KUKA KRL program: MyProgram_236().src

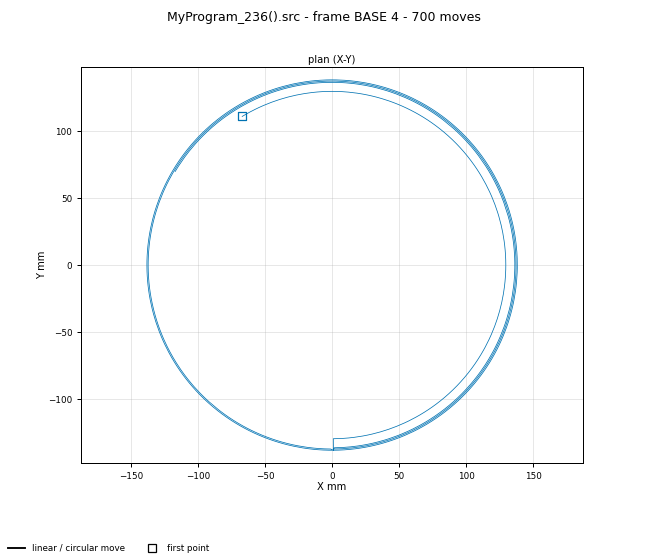
[picture p0: tool path of MyProgram_236().src in frame BASE 4, 700 of 700 moves have a stored position in this frame; points joined in program order, loops and branches not executed]
&ACCESS RVP
&REL 1
&PARAM TEMPLATE = C:\KRC\Roboter\Template\vorgabe
&PARAM EDITMASK = *
DEF MyProgram_236()
; ---- Setting reference (Base) ----
$BASE = BASE_DATA[4]

; --------------------------
; ---- Setting tool (TCP) ----
$TOOL = TOOL_DATA[3]
; --------------------------

$VEL.CP = VEL_APROX_PRINT
Startdeposition()
$VEL.CP = VEL_PRINT
LIN {X -67.1203,Y 110.906,Z 159,A 119.8664,B 14.7738,C -0.2462,E1 14.6942,E2 329.6728} C_DIS
LIN {X -63.8698,Y 112.81,Z 159,A 118.1875,B 14.7738,C -0.2484,E1 14.6982,E2 331.3516} C_DIS
LIN {X -61.0916,Y 114.338,Z 159,A 116.7775,B 14.7738,C -0.2503,E1 14.7017,E2 332.7612} C_DIS
LIN {X -57.3512,Y 116.2566,Z 159,A 114.9162,B 14.7737,C -0.2529,E1 14.7063,E2 334.6209} C_DIS
LIN {X -54.4896,Y 117.6251,Z 159,A 113.4128,B 14.7737,C -0.2521,E1 14.7102,E2 336.1345} C_DIS
LIN {X -51.0857,Y 119.1435,Z 159,A 111.8471,B 14.7737,C -0.2564,E1 14.7141,E2 337.6895} C_DIS
LIN {X -48.1337,Y 120.3663,Z 159,A 110.4314,B 14.7736,C -0.2581,E1 14.7178,E2 339.1043} C_DIS
LIN {X -45.1664,Y 121.5109,Z 159,A 109.0181,B 14.7736,C -0.2595,E1 14.7215,E2 340.5173} C_DIS
LIN {X -42.1522,Y 122.5891,Z 159,A 107.6016,B 14.7736,C -0.261,E1 14.7252,E2 341.9327} C_DIS
LIN {X -39.1386,Y 123.5843,Z 159,A 106.1946,B 14.7736,C -0.2623,E1 14.7289,E2 343.3391} C_DIS
LIN {X -36.1004,Y 124.5058,Z 159,A 104.7875,B 14.7736,C -0.2635,E1 14.7327,E2 344.7455} C_DIS
LIN {X -33.0403,Y 125.3527,Z 159,A 103.3786,B 14.7735,C -0.2646,E1 14.7365,E2 346.1539} C_DIS
LIN {X -29.9406,Y 126.1293,Z 159,A 101.9667,B 14.7735,C -0.2657,E1 14.7403,E2 347.5647} C_DIS
LIN {X -26.8488,Y 126.8237,Z 159,A 100.5599,B 14.7735,C -0.2665,E1 14.7442,E2 348.9712} C_DIS
LIN {X -24.2125,Y 127.3523,Z 159,A 99.3725,B 14.7735,C -0.2674,E1 14.7474,E2 350.1576} C_DIS
LIN {X -20.8059,Y 127.9541,Z 159,A 97.868,B 14.7735,C -0.269,E1 14.7516,E2 351.6584} C_DIS
LIN {X -18.0217,Y 128.3752,Z 159,A 96.6198,B 14.7734,C -0.2695,E1 14.755,E2 352.9061} C_DIS
LIN {X -14.8341,Y 128.7831,Z 159,A 95.0397,B 14.7734,C -0.2656,E1 14.7594,E2 354.5036} C_DIS
LIN {X -11.1216,Y 129.1559,Z 159,A 93.509,B 14.7734,C -0.2696,E1 14.7636,E2 356.0199} C_DIS
LIN {X -7.5683,Y 129.4132,Z 159,A 91.939,B 14.7734,C -0.2702,E1 14.768,E2 357.5884} C_DIS
LIN {X -3.731,Y 129.5801,Z 159,A 90.2362,B 14.7734,C -0.2704,E1 14.7728,E2 359.2909} C_DIS
LIN {X 0.0023,Y 129.6358,Z 159,A 88.562,B 14.7734,C -0.2699,E1 14.7774,E2 360.9671} C_DIS
LIN {X 3.733,Y 129.5801,Z 159,A 86.8871,B 14.7734,C -0.2692,E1 14.7821,E2 362.6441} C_DIS
LIN {X 7.9541,Y 129.3894,Z 159,A 84.9994,B 14.7734,C -0.2685,E1 14.7874,E2 364.5334} C_DIS
LIN {X 12.1572,Y 129.0626,Z 159,A 83.138,B 14.7734,C -0.2682,E1 14.7926,E2 366.3939} C_DIS
LIN {X 16.0012,Y 128.6439,Z 159,A 81.5164,B 14.7734,C -0.2703,E1 14.797,E2 368.005} C_DIS
LIN {X 18.6052,Y 128.2918,Z 159,A 80.3418,B 14.7734,C -0.2696,E1 14.8003,E2 369.1807} C_DIS
LIN {X 22.1957,Y 127.7209,Z 159,A 78.5869,B 14.7734,C -0.2645,E1 14.8052,E2 370.9521} C_DIS
LIN {X 26.3286,Y 126.9326,Z 159,A 76.8852,B 14.7734,C -0.2683,E1 14.8098,E2 372.6354} C_DIS
LIN {X 29.4247,Y 126.2511,Z 159,A 75.486,B 14.7734,C -0.2676,E1 14.8136,E2 374.0341} C_DIS
LIN {X 33.0382,Y 125.3533,Z 159,A 73.7666,B 14.7734,C -0.2643,E1 14.8183,E2 375.7616} C_DIS
LIN {X 37.1039,Y 124.212,Z 159,A 71.979,B 14.7734,C -0.2653,E1 14.823,E2 377.5401} C_DIS
LIN {X 40.1416,Y 123.2639,Z 159,A 70.5796,B 14.7734,C -0.2643,E1 14.8268,E2 378.9385} C_DIS
LIN {X 42.6971,Y 122.4002,Z 159,A 69.3347,B 14.7735,C -0.2617,E1 14.8301,E2 380.1893} C_DIS
LIN {X 45.6848,Y 121.3167,Z 159,A 67.9319,B 14.7735,C -0.2604,E1 14.8337,E2 381.5919} C_DIS
LIN {X 49.089,Y 119.9813,Z 159,A 66.3714,B 14.7735,C -0.2604,E1 14.8378,E2 383.146} C_DIS
LIN {X 52.0319,Y 118.7345,Z 159,A 64.8389,B 14.7736,C -0.2552,E1 14.8417,E2 384.6923} C_DIS
LIN {X 55.4342,Y 117.1839,Z 159,A 63.328,B 14.7736,C -0.2576,E1 14.8455,E2 386.1871} C_DIS
LIN {X 58.7836,Y 115.539,Z 159,A 61.6551,B 14.7736,C -0.2548,E1 14.8497,E2 387.8628} C_DIS
LIN {X 62.0192,Y 113.8372,Z 159,A 60.0736,B 14.7736,C -0.2537,E1 14.8536,E2 389.4408} C_DIS
LIN {X 64.7903,Y 112.2832,Z 159,A 58.5716,B 14.7738,C -0.2487,E1 14.8573,E2 390.9543} C_DIS
LIN {X 68.0623,Y 110.3309,Z 159,A 56.8912,B 14.7738,C -0.2463,E1 14.8613,E2 392.6346} C_DIS
LIN {X 71.5703,Y 108.0883,Z 159,A 55.1642,B 14.7738,C -0.2469,E1 14.8653,E2 394.3491} C_DIS
LIN {X 74.1944,Y 106.3038,Z 159,A 53.7715,B 14.7738,C -0.2449,E1 14.8685,E2 395.7411} C_DIS
LIN {X 77.2242,Y 104.1238,Z 159,A 51.9984,B 14.7739,C -0.2383,E1 14.8725,E2 397.529} C_DIS
LIN {X 80.4688,Y 101.6374,Z 159,A 50.1936,B 14.7739,C -0.2352,E1 14.8765,E2 399.3342} C_DIS
LIN {X 83.8675,Y 98.8511,Z 159,A 48.359,B 14.7739,C -0.2349,E1 14.8804,E2 401.1572} C_DIS
LIN {X 86.6751,Y 96.399,Z 159,A 46.6678,B 14.774,C -0.2304,E1 14.884,E2 402.8541} C_DIS
LIN {X 89.7611,Y 93.5323,Z 159,A 44.8758,B 14.774,C -0.2289,E1 14.8876,E2 404.639} C_DIS
LIN {X 92.742,Y 90.5774,Z 159,A 42.9905,B 14.7741,C -0.2241,E1 14.8913,E2 406.5288} C_DIS
LIN {X 95.5533,Y 87.6064,Z 159,A 41.2364,B 14.7741,C -0.2219,E1 14.8946,E2 408.2777} C_DIS
LIN {X 98.3326,Y 84.4748,Z 159,A 39.347,B 14.7742,C -0.2166,E1 14.8981,E2 410.1727} C_DIS
LIN {X 101.04,Y 81.2173,Z 159,A 37.4829,B 14.7743,C -0.2127,E1 14.9014,E2 412.0371} C_DIS
LIN {X 103.7073,Y 77.7832,Z 159,A 35.5408,B 14.7743,C -0.2075,E1 14.9047,E2 413.9828} C_DIS
LIN {X 105.9847,Y 74.6493,Z 159,A 33.989,B 14.7743,C -0.2086,E1 14.9072,E2 415.5174} C_DIS
LIN {X 107.7826,Y 72.0291,Z 159,A 32.599,B 14.7744,C -0.2056,E1 14.9094,E2 416.9066} C_DIS
LIN {X 109.8271,Y 68.8726,Z 159,A 30.8417,B 14.7744,C -0.1984,E1 14.912,E2 418.6763} C_DIS
LIN {X 111.7248,Y 65.7484,Z 159,A 29.2525,B 14.7745,C -0.1952,E1 14.9143,E2 420.2637} C_DIS
LIN {X 113.5698,Y 62.5083,Z 159,A 27.7539,B 14.7745,C -0.1958,E1 14.9163,E2 421.7464} C_DIS
LIN {X 114.8093,Y 60.1962,Z 159,A 26.5652,B 14.7745,C -0.1918,E1 14.9179,E2 422.9394} C_DIS
LIN {X 116.2491,Y 57.3666,Z 159,A 25.1756,B 14.7746,C -0.1885,E1 14.9196,E2 424.3286} C_DIS
LIN {X 117.6203,Y 54.5,Z 159,A 23.6885,B 14.7747,C -0.1821,E1 14.9214,E2 425.8266} C_DIS
LIN {X 119.1501,Y 51.0705,Z 159,A 22.1376,B 14.7747,C -0.1811,E1 14.9231,E2 427.3664} C_DIS
LIN {X 120.3664,Y 48.1335,Z 159,A 20.7467,B 14.7747,C -0.1777,E1 14.9246,E2 428.757} C_DIS
LIN {X 121.5105,Y 45.1674,Z 159,A 19.3557,B 14.7747,C -0.1743,E1 14.926,E2 430.1477} C_DIS
LIN {X 122.5834,Y 42.1688,Z 159,A 17.9628,B 14.7748,C -0.1708,E1 14.9273,E2 431.5403} C_DIS
LIN {X 123.5841,Y 39.1391,Z 159,A 16.5673,B 14.7748,C -0.1673,E1 14.9285,E2 432.9355} C_DIS
LIN {X 124.4063,Y 36.44,Z 159,A 15.2755,B 14.7749,C -0.1623,E1 14.9295,E2 434.2338} C_DIS
LIN {X 125.3524,Y 33.0414,Z 159,A 13.7909,B 14.7749,C -0.1602,E1 14.9306,E2 435.7114} C_DIS
LIN {X 126.124,Y 29.9624,Z 159,A 12.4206,B 14.7749,C -0.1572,E1 14.9315,E2 437.0794} C_DIS
LIN {X 126.8601,Y 26.6802,Z 159,A 10.9379,B 14.775,C -0.153,E1 14.9324,E2 438.5633} C_DIS
LIN {X 127.3533,Y 24.2074,Z 159,A 9.8335,B 14.775,C -0.1501,E1 14.933,E2 439.6677} C_DIS
LIN {X 127.9849,Y 20.6214,Z 159,A 8.2534,B 14.775,C -0.1462,E1 14.9337,E2 441.2463} C_DIS
LIN {X 128.3792,Y 17.9938,Z 159,A 7.0773,B 14.7751,C -0.1427,E1 14.9342,E2 442.4238} C_DIS
LIN {X 128.7823,Y 14.841,Z 159,A 5.5559,B 14.7751,C -0.1347,E1 14.9347,E2 443.9605} C_DIS
LIN {X 129.1554,Y 11.1276,Z 159,A 3.9869,B 14.7752,C -0.1324,E1 14.9351,E2 445.522} C_DIS
LIN {X 129.4343,Y 7.2235,Z 159,A 2.3652,B 14.7752,C -0.1308,E1 14.9354,E2 447.1332} C_DIS
LIN {X 129.5799,Y 3.7378,Z 159,A 0.8063,B 14.7752,C -0.1256,E1 14.9356,E2 448.6959} C_DIS
LIN {X 129.636,Y 0.0053,Z 159,A -0.8546,B 14.7753,C -0.1202,E1 14.9356,E2 450.3602} C_DIS
LIN {X 129.5905,Y -3.3568,Z 159,A -2.4308,B 14.7753,C -0.1128,E1 14.9356,E2 451.9486} C_DIS
LIN {X 129.3897,Y -7.9495,Z 159,A -4.3756,B 14.7754,C -0.1096,E1 14.9352,E2 453.8858} C_DIS
LIN {X 129.0632,Y -12.1507,Z 159,A -6.1534,B 14.7754,C -0.1067,E1 14.9348,E2 455.656} C_DIS
LIN {X 128.6351,Y -16.0754,Z 159,A -7.8536,B 14.7754,C -0.1029,E1 14.9343,E2 457.3533} C_DIS
LIN {X 128.2236,Y -19.0827,Z 159,A -9.2075,B 14.7754,C -0.0985,E1 14.9337,E2 458.7104} C_DIS
LIN {X 127.8138,Y -21.6469,Z 159,A -10.418,B 14.7755,C -0.093,E1 14.9332,E2 459.9295} C_DIS
LIN {X 127.1942,Y -25.0399,Z 159,A -11.8339,B 14.7755,C -0.092,E1 14.9324,E2 461.3348} C_DIS
LIN {X 126.6015,Y -27.8778,Z 159,A -13.11,B 14.7755,C -0.0884,E1 14.9317,E2 462.6119} C_DIS
LIN {X 125.9172,Y -30.8204,Z 159,A -14.4371,B 14.7755,C -0.0847,E1 14.9308,E2 463.9398} C_DIS
LIN {X 125.0892,Y -34.0284,Z 159,A -15.8607,B 14.7755,C -0.0817,E1 14.9298,E2 465.3605} C_DIS
LIN {X 124.2104,Y -37.1093,Z 159,A -17.2862,B 14.7756,C -0.0772,E1 14.9287,E2 466.789} C_DIS
LIN {X 123.2639,Y -40.1415,Z 159,A -18.6777,B 14.7756,C -0.0736,E1 14.9275,E2 468.1808} C_DIS
LIN {X 122.4011,Y -42.6947,Z 159,A -19.9406,B 14.7756,C -0.0678,E1 14.9264,E2 469.4537} C_DIS
LIN {X 121.282,Y -45.7774,Z 159,A -21.336,B 14.7756,C -0.0654,E1 14.925,E2 470.8447} C_DIS
LIN {X 119.9587,Y -49.145,Z 159,A -22.8797,B 14.7756,C -0.0626,E1 14.9234,E2 472.3841} C_DIS
LIN {X 118.8209,Y -51.8319,Z 159,A -24.1799,B 14.7756,C -0.0587,E1 14.922,E2 473.6871} C_DIS
LIN {X 117.1943,Y -55.4124,Z 159,A -25.8759,B 14.7756,C -0.0552,E1 14.92,E2 475.3804} C_DIS
LIN {X 115.7914,Y -58.2877,Z 159,A -27.2678,B 14.7757,C -0.052,E1 14.9183,E2 476.7716} C_DIS
LIN {X 114.3285,Y -61.1093,Z 159,A -28.5712,B 14.7757,C -0.0515,E1 14.9166,E2 478.0649} C_DIS
LIN {X 113.0667,Y -63.413,Z 159,A -29.9152,B 14.7757,C -0.0423,E1 14.9147,E2 479.432} C_DIS
LIN {X 110.8982,Y -67.1332,Z 159,A -31.7839,B 14.7757,C -0.0384,E1 14.9121,E2 481.2991} C_DIS
LIN {X 108.6614,Y -70.6965,Z 159,A -33.5454,B 14.7757,C -0.0367,E1 14.9095,E2 483.0515} C_DIS
LIN {X 106.5523,Y -73.8374,Z 159,A -35.2973,B 14.7757,C -0.0298,E1 14.9067,E2 484.8149} C_DIS
LIN {X 104.1116,Y -77.2405,Z 159,A -37.1373,B 14.7757,C -0.0255,E1 14.9037,E2 486.656} C_DIS
LIN {X 101.5297,Y -80.6041,Z 159,A -38.9905,B 14.7757,C -0.0216,E1 14.9005,E2 488.5091} C_DIS
LIN {X 98.8199,Y -83.9042,Z 159,A -40.8594,B 14.7757,C -0.0176,E1 14.8971,E2 490.3782} C_DIS
LIN {X 96.0345,Y -87.0784,Z 159,A -42.7041,B 14.7757,C -0.014,E1 14.8937,E2 492.2226} C_DIS
LIN {X 93.3312,Y -89.9702,Z 159,A -44.4989,B 14.7757,C -0.0085,E1 14.8902,E2 494.0249} C_DIS
LIN {X 90.133,Y -93.1735,Z 159,A -46.4359,B 14.7757,C -0.0061,E1 14.8864,E2 495.9568} C_DIS
LIN {X 87.0427,Y -96.0669,Z 159,A -48.287,B 14.7758,C -0.0027,E1 14.8826,E2 497.8078} C_DIS
LIN {X 84.0655,Y -98.6827,Z 159,A -49.989,B 14.7758,C -0.0007,E1 14.879,E2 499.506} C_DIS
LIN {X 80.9868,Y -101.2251,Z 159,A -51.8385,B 14.7758,C 0.0056,E1 14.875,E2 501.3675} C_DIS
LIN {X 77.6558,Y -103.8024,Z 159,A -53.6478,B 14.7758,C 0.0076,E1 14.871,E2 503.1727} C_DIS
LIN {X 74.6416,Y -105.9902,Z 159,A -55.1713,B 14.7758,C 0.0067,E1 14.8675,E2 504.6837} C_DIS
LIN {X 72.0229,Y -107.7867,Z 159,A -56.5633,B 14.7758,C 0.0089,E1 14.8643,E2 506.0757} C_DIS
LIN {X 68.9171,Y -109.799,Z 159,A -58.3045,B 14.7758,C 0.0151,E1 14.8602,E2 507.8312} C_DIS
LIN {X 65.7525,Y -111.7224,Z 159,A -59.896,B 14.7758,C 0.0164,E1 14.8564,E2 509.4191} C_DIS
LIN {X 62.5084,Y -113.5697,Z 159,A -61.4627,B 14.7758,C 0.0164,E1 14.8526,E2 510.9776} C_DIS
LIN {X 59.5138,Y -115.1672,Z 159,A -62.9484,B 14.7758,C 0.0183,E1 14.8489,E2 512.4632} C_DIS
LIN {X 57.2074,Y -116.3276,Z 159,A -64.0735,B 14.7758,C 0.0195,E1 14.8461,E2 513.5874} C_DIS
LIN {X 54.0617,Y -117.8229,Z 159,A -65.6278,B 14.7758,C 0.0221,E1 14.8422,E2 515.145} C_DIS
LIN {X 51.0647,Y -119.1526,Z 159,A -67.0629,B 14.7758,C 0.0236,E1 14.8385,E2 516.5798} C_DIS
LIN {X 48.1302,Y -120.3678,Z 159,A -68.4596,B 14.7758,C 0.0252,E1 14.8349,E2 517.9769} C_DIS
LIN {X 45.1639,Y -121.5118,Z 159,A -69.8579,B 14.7758,C 0.0267,E1 14.8312,E2 519.3757} C_DIS
LIN {X 42.1715,Y -122.5825,Z 159,A -71.2646,B 14.7758,C 0.0283,E1 14.8275,E2 520.7837} C_DIS
LIN {X 39.097,Y -123.5976,Z 159,A -72.6797,B 14.7758,C 0.0294,E1 14.8237,E2 522.1982} C_DIS
LIN {X 36.0775,Y -124.5125,Z 159,A -74.0689,B 14.7758,C 0.0306,E1 14.82,E2 523.588} C_DIS
LIN {X 33.0288,Y -125.3558,Z 159,A -75.4487,B 14.7758,C 0.0314,E1 14.8163,E2 524.9666} C_DIS
LIN {X 29.9586,Y -126.1249,Z 159,A -76.8546,B 14.7758,C 0.0328,E1 14.8125,E2 526.3745} C_DIS
LIN {X 26.3447,Y -126.9293,Z 159,A -78.5984,B 14.7758,C 0.0374,E1 14.8077,E2 528.1321} C_DIS
LIN {X 22.7058,Y -127.6296,Z 159,A -80.1843,B 14.7758,C 0.0369,E1 14.8034,E2 529.713} C_DIS
LIN {X 19.5724,Y -128.1478,Z 159,A -81.5205,B 14.7758,C 0.0357,E1 14.7997,E2 531.0423} C_DIS
LIN {X 16.4157,Y -128.5908,Z 159,A -83.0436,B 14.7758,C 0.04,E1 14.7954,E2 532.5797} C_DIS
LIN {X 12.1492,Y -129.0633,Z 159,A -84.886,B 14.7758,C 0.0392,E1 14.7903,E2 534.4168} C_DIS
LIN {X 7.9488,Y -129.3898,Z 159,A -86.7504,B 14.7758,C 0.0399,E1 14.7851,E2 536.2825} C_DIS
LIN {X 3.7245,Y -129.5803,Z 159,A -88.5546,B 14.7758,C 0.0385,E1 14.7801,E2 538.0802} C_DIS
LIN {X 0.8939,Y -129.6275,Z 159,A -89.3751,B 14.7758,C 0.0257,E1 14.778,E2 538.8503} C_DIS
Enddeposition()
LIN {X 0.9745,Y -138.2214,Z 160,A -92.2372,B 24.9707,C -1.2506,E1 25.0023,E2 538.9144} C_DIS
Startdeposition()
$VEL.CP = VEL_PRINT
LIN {X 4.9672,Y -138.1363,Z 160,A -90.5146,B 24.9705,C -1.2549,E1 25.0072,E2 537.182} C_DIS
LIN {X 8.9652,Y -137.9346,Z 160,A -88.7661,B 24.9702,C -1.2605,E1 25.0121,E2 535.4208} C_DIS
LIN {X 12.9848,Y -137.6138,Z 160,A -87.2521,B 24.9706,C -1.2526,E1 25.0162,E2 533.9264} C_DIS
LIN {X 17.0609,Y -137.1696,Z 160,A -85.4986,B 24.9704,C -1.2567,E1 25.0211,E2 532.1646} C_DIS
LIN {X 20.739,Y -136.6607,Z 160,A -83.946,B 24.9704,C -1.2585,E1 25.0254,E2 530.609} C_DIS
LIN {X 24.3768,Y -136.0582,Z 160,A -82.4644,B 24.9704,C -1.2571,E1 25.0295,E2 529.1323} C_DIS
LIN {X 27.7328,Y -135.4141,Z 160,A -81.0374,B 24.9704,C -1.259,E1 25.0334,E2 527.7026} C_DIS
LIN {X 31.1838,Y -134.6618,Z 160,A -79.4483,B 24.9699,C -1.2674,E1 25.0378,E2 526.0957} C_DIS
LIN {X 34.8431,Y -133.7633,Z 160,A -78.028,B 24.9702,C -1.261,E1 25.0416,E2 524.6926} C_DIS
LIN {X 38.2167,Y -132.838,Z 160,A -76.5857,B 24.9702,C -1.2622,E1 25.0455,E2 523.25} C_DIS
LIN {X 41.4498,Y -131.8649,Z 160,A -75.1438,B 24.97,C -1.2663,E1 25.0493,E2 521.801} C_DIS
LIN {X 44.7534,Y -130.7801,Z 160,A -73.6382,B 24.9697,C -1.2718,E1 25.0533,E2 520.2853} C_DIS
LIN {X 48.3409,Y -129.4959,Z 160,A -72.1957,B 24.97,C -1.2662,E1 25.0571,E2 518.8591} C_DIS
LIN {X 51.4463,Y -128.294,Z 160,A -70.8247,B 24.97,C -1.2676,E1 25.0606,E2 517.4876} C_DIS
LIN {X 54.8596,Y -126.8716,Z 160,A -69.2999,B 24.9698,C -1.2695,E1 25.0646,E2 515.962} C_DIS
LIN {X 57.9395,Y -125.495,Z 160,A -67.8796,B 24.9697,C -1.273,E1 25.0682,E2 514.5371} C_DIS
LIN {X 60.4907,Y -124.2875,Z 160,A -66.6861,B 24.9695,C -1.2762,E1 25.0712,E2 513.3391} C_DIS
LIN {X 63.6062,Y -122.7223,Z 160,A -65.2643,B 24.9695,C -1.2774,E1 25.0747,E2 511.9184} C_DIS
LIN {X 66.6673,Y -121.0872,Z 160,A -63.7025,B 24.969,C -1.287,E1 25.0786,E2 510.3384} C_DIS
LIN {X 70.4482,Y -118.9273,Z 160,A -61.8999,B 24.9688,C -1.2903,E1 25.083,E2 508.5336} C_DIS
LIN {X 74.2885,Y -116.5668,Z 160,A -60.0462,B 24.9687,C -1.2931,E1 25.0873,E2 506.6792} C_DIS
LIN {X 77.8899,Y -114.1921,Z 160,A -58.3083,B 24.9687,C -1.2938,E1 25.0914,E2 504.9453} C_DIS
LIN {X 81.4971,Y -111.6464,Z 160,A -56.5752,B 24.9687,C -1.2921,E1 25.0953,E2 503.2223} C_DIS
LIN {X 84.31,Y -109.5377,Z 160,A -54.9752,B 24.9682,C -1.3036,E1 25.0989,E2 501.6011} C_DIS
LIN {X 87.8225,Y -106.7423,Z 160,A -53.1459,B 24.9681,C -1.306,E1 25.1028,E2 499.773} C_DIS
LIN {X 91.2002,Y -103.8712,Z 160,A -51.2962,B 24.9678,C -1.311,E1 25.1068,E2 497.9188} C_DIS
LIN {X 94.3975,Y -100.9737,Z 160,A -49.6476,B 24.968,C -1.3073,E1 25.1101,E2 496.2857} C_DIS
LIN {X 97.053,Y -98.4244,Z 160,A -48.142,B 24.9679,C -1.3099,E1 25.1131,E2 494.7802} C_DIS
LIN {X 99.5318,Y -95.9169,Z 160,A -46.6892,B 24.9677,C -1.3131,E1 25.116,E2 493.3261} C_DIS
LIN {X 101.9451,Y -93.3477,Z 160,A -45.2383,B 24.9675,C -1.3163,E1 25.1187,E2 491.874} C_DIS
LIN {X 104.2139,Y -90.8074,Z 160,A -43.7946,B 24.9673,C -1.3219,E1 25.1214,E2 490.4236} C_DIS
LIN {X 106.6121,Y -87.9797,Z 160,A -42.291,B 24.9672,C -1.3241,E1 25.1241,E2 488.9217} C_DIS
LIN {X 108.8159,Y -85.2388,Z 160,A -40.858,B 24.967,C -1.3267,E1 25.1266,E2 487.4893} C_DIS
LIN {X 110.943,Y -82.4511,Z 160,A -39.414,B 24.9669,C -1.3302,E1 25.129,E2 486.044} C_DIS
LIN {X 113.1108,Y -79.4515,Z 160,A -37.8654,B 24.9666,C -1.3354,E1 25.1315,E2 484.4905} C_DIS
LIN {X 115.116,Y -76.5173,Z 160,A -36.4114,B 24.9664,C -1.3385,E1 25.1338,E2 483.0364} C_DIS
LIN {X 117.4083,Y -72.9508,Z 160,A -34.6661,B 24.9662,C -1.343,E1 25.1364,E2 481.2895} C_DIS
LIN {X 119.2406,Y -69.9157,Z 160,A -33.2242,B 24.9661,C -1.3457,E1 25.1384,E2 479.8484} C_DIS
LIN {X 121.2665,Y -66.34,Z 160,A -31.487,B 24.9657,C -1.3528,E1 25.1408,E2 478.1035} C_DIS
LIN {X 123.0416,Y -62.9827,Z 160,A -29.9644,B 24.9657,C -1.3547,E1 25.1428,E2 476.5846} C_DIS
LIN {X 124.5999,Y -59.8407,Z 160,A -28.4957,B 24.9654,C -1.36,E1 25.1446,E2 475.1112} C_DIS
LIN {X 126.1424,Y -56.5163,Z 160,A -27.0475,B 24.9654,C -1.3606,E1 25.1463,E2 473.6694} C_DIS
LIN {X 127.6265,Y -53.0803,Z 160,A -25.4802,B 24.965,C -1.3664,E1 25.148,E2 472.0971} C_DIS
LIN {X 128.8893,Y -49.9357,Z 160,A -24.0757,B 24.9648,C -1.3709,E1 25.1494,E2 470.6898} C_DIS
LIN {X 130.0588,Y -46.805,Z 160,A -22.6836,B 24.9645,C -1.3757,E1 25.1507,E2 469.2942} C_DIS
LIN {X 131.2188,Y -43.4477,Z 160,A -21.2376,B 24.9644,C -1.3789,E1 25.152,E2 467.8487} C_DIS
LIN {X 132.3059,Y -40.0173,Z 160,A -19.7444,B 24.9641,C -1.3838,E1 25.1533,E2 466.3524} C_DIS
LIN {X 133.283,Y -36.6339,Z 160,A -18.3051,B 24.9639,C -1.3874,E1 25.1544,E2 464.9131} C_DIS
LIN {X 134.174,Y -33.2269,Z 160,A -16.8522,B 24.9637,C -1.3917,E1 25.1554,E2 463.4583} C_DIS
LIN {X 134.9761,Y -29.7979,Z 160,A -15.3929,B 24.9635,C -1.3965,E1 25.1563,E2 461.9961} C_DIS
LIN {X 135.6701,Y -26.4563,Z 160,A -13.961,B 24.9632,C -1.4022,E1 25.1571,E2 460.5591} C_DIS
LIN {X 136.3134,Y -22.9074,Z 160,A -12.6947,B 24.9636,C -1.3938,E1 25.1577,E2 459.3201} C_DIS
LIN {X 136.7952,Y -19.8301,Z 160,A -11.2092,B 24.9628,C -1.4095,E1 25.1583,E2 457.8065} C_DIS
LIN {X 137.2552,Y -16.3433,Z 160,A -9.7726,B 24.9626,C -1.4131,E1 25.1588,E2 456.3698} C_DIS
LIN {X 137.6767,Y -12.3167,Z 160,A -8.1609,B 24.9626,C -1.4148,E1 25.1592,E2 454.7637} C_DIS
LIN {X 137.9473,Y -8.7588,Z 160,A -6.6567,B 24.9622,C -1.4212,E1 25.1595,E2 453.2534} C_DIS
LIN {X 138.1179,Y -5.4374,Z 160,A -5.2669,B 24.9619,C -1.4264,E1 25.1597,E2 451.8594} C_DIS
LIN {X 138.2105,Y -2.0186,Z 160,A -3.9101,B 24.9619,C -1.4276,E1 25.1597,E2 450.508} C_DIS
LIN {X 138.209,Y 2.1074,Z 160,A -2.0773,B 24.9611,C -1.4405,E1 25.1597,E2 448.6557} C_DIS
LIN {X 138.1274,Y 5.1947,Z 160,A -0.6881,B 24.9606,C -1.4511,E1 25.1597,E2 447.2498} C_DIS
LIN {X 137.8703,Y 9.8947,Z 160,A 0.9764,B 24.9611,C -1.4408,E1 25.1593,E2 445.6195} C_DIS
LIN {X 137.5862,Y 13.2721,Z 160,A 2.2425,B 24.9613,C -1.4373,E1 25.159,E2 444.369} C_DIS
LIN {X 137.2722,Y 16.2009,Z 160,A 3.6087,B 24.9606,C -1.4498,E1 25.1586,E2 442.9816} C_DIS
LIN {X 136.8421,Y 19.5022,Z 160,A 5.0189,B 24.9603,C -1.456,E1 25.158,E2 441.5649} C_DIS
LIN {X 136.318,Y 22.8797,Z 160,A 6.4378,B 24.96,C -1.4608,E1 25.1574,E2 440.1432} C_DIS
LIN {X 135.6895,Y 26.3551,Z 160,A 7.882,B 24.9598,C -1.4643,E1 25.1567,E2 438.699} C_DIS
LIN {X 134.9428,Y 29.9523,Z 160,A 9.3918,B 24.9596,C -1.4684,E1 25.1558,E2 437.1884} C_DIS
LIN {X 134.1367,Y 33.3737,Z 160,A 10.8442,B 24.9594,C -1.4728,E1 25.1548,E2 435.7341} C_DIS
LIN {X 133.2441,Y 36.7732,Z 160,A 12.29,B 24.9591,C -1.4768,E1 25.1538,E2 434.2873} C_DIS
LIN {X 132.1998,Y 40.364,Z 160,A 13.822,B 24.9589,C -1.4806,E1 25.1526,E2 432.755} C_DIS
LIN {X 130.8683,Y 44.4992,Z 160,A 15.6087,B 24.9587,C -1.4853,E1 25.151,E2 430.9673} C_DIS
LIN {X 129.7193,Y 47.7444,Z 160,A 17.0621,B 24.9583,C -1.4912,E1 25.1496,E2 429.5082} C_DIS
LIN {X 128.531,Y 50.8572,Z 160,A 18.4196,B 24.9582,C -1.494,E1 25.1482,E2 428.1516} C_DIS
LIN {X 127.0386,Y 54.4733,Z 160,A 19.9763,B 24.9582,C -1.4951,E1 25.1466,E2 426.6008} C_DIS
LIN {X 125.7091,Y 57.4765,Z 160,A 21.4262,B 24.9576,C -1.5042,E1 25.1449,E2 425.1373} C_DIS
LIN {X 124.1173,Y 60.8357,Z 160,A 22.8957,B 24.9576,C -1.5046,E1 25.1431,E2 423.6749} C_DIS
LIN {X 122.5419,Y 63.9498,Z 160,A 24.2901,B 24.9576,C -1.5057,E1 25.1413,E2 422.2851} C_DIS
LIN {X 120.9445,Y 66.925,Z 160,A 25.8014,B 24.9569,C -1.5161,E1 25.1393,E2 420.7574} C_DIS
LIN {X 118.7599,Y 70.7292,Z 160,A 27.5663,B 24.9569,C -1.518,E1 25.1368,E2 418.997} C_DIS
LIN {X 116.8423,Y 73.8539,Z 160,A 29.1851,B 24.9563,C -1.5278,E1 25.1344,E2 417.3632} C_DIS
LIN {X 114.3131,Y 77.7117,Z 160,A 30.9658,B 24.9564,C -1.5253,E1 25.1316,E2 415.5973} C_DIS
LIN {X 111.8821,Y 81.1721,Z 160,A 32.7079,B 24.9562,C -1.5292,E1 25.1288,E2 413.8544} C_DIS
LIN {X 109.8325,Y 83.9247,Z 160,A 34.1226,B 24.956,C -1.5324,E1 25.1264,E2 412.439} C_DIS
LIN {X 107.5881,Y 86.7832,Z 160,A 35.63,B 24.9558,C -1.5362,E1 25.1238,E2 410.9298} C_DIS
LIN {X 105.34,Y 89.4986,Z 160,A 37.1424,B 24.9554,C -1.5426,E1 25.1211,E2 409.409} C_DIS
LIN {X 102.4288,Y 92.8163,Z 160,A 38.8997,B 24.9554,C -1.5428,E1 25.1178,E2 407.6592} C_DIS
LIN {X 99.5239,Y 95.925,Z 160,A 40.6801,B 24.9551,C -1.5477,E1 25.1144,E2 405.8748} C_DIS
LIN {X 96.8304,Y 98.6428,Z 160,A 42.2116,B 24.9551,C -1.5481,E1 25.1114,E2 404.3489} C_DIS
LIN {X 94.3231,Y 101.043,Z 160,A 43.7287,B 24.9547,C -1.5556,E1 25.1083,E2 402.8203} C_DIS
LIN {X 91.0837,Y 103.9728,Z 160,A 45.512,B 24.9545,C -1.5578,E1 25.1046,E2 401.039} C_DIS
LIN {X 88.2077,Y 106.4233,Z 160,A 47.0049,B 24.9545,C -1.5568,E1 25.1014,E2 399.5542} C_DIS
LIN {X 85.2684,Y 108.7926,Z 160,A 48.6625,B 24.9541,C -1.565,E1 25.0977,E2 397.8835} C_DIS
LIN {X 82.1688,Y 111.1529,Z 160,A 50.1778,B 24.9543,C -1.5623,E1 25.0944,E2 396.38} C_DIS
LIN {X 79.2048,Y 113.2838,Z 160,A 51.684,B 24.9541,C -1.5646,E1 25.0909,E2 394.8736} C_DIS
LIN {X 76.2691,Y 115.2807,Z 160,A 53.1264,B 24.9541,C -1.5654,E1 25.0876,E2 393.4341} C_DIS
LIN {X 73.3175,Y 117.1801,Z 160,A 54.7133,B 24.9535,C -1.5752,E1 25.0838,E2 391.8293} C_DIS
LIN {X 69.5028,Y 119.4821,Z 160,A 56.5806,B 24.9533,C -1.5792,E1 25.0793,E2 389.9583} C_DIS
LIN {X 65.7681,Y 121.5781,Z 160,A 58.3047,B 24.9533,C -1.5788,E1 25.0751,E2 388.24} C_DIS
LIN {X 62.7743,Y 123.1477,Z 160,A 59.4484,B 24.954,C -1.5664,E1 25.0724,E2 387.1289} C_DIS
LIN {X 60.2,Y 124.4283,Z 160,A 60.8337,B 24.9533,C -1.5786,E1 25.0688,E2 385.7183} C_DIS
LIN {X 56.9939,Y 125.9287,Z 160,A 62.2678,B 24.9533,C -1.5786,E1 25.0652,E2 384.288} C_DIS
LIN {X 53.7648,Y 127.3406,Z 160,A 63.7726,B 24.9531,C -1.5827,E1 25.0613,E2 382.777} C_DIS
LIN {X 50.358,Y 128.7251,Z 160,A 65.3418,B 24.9528,C -1.5868,E1 25.0572,E2 381.2016} C_DIS
LIN {X 46.3964,Y 130.2062,Z 160,A 67.0041,B 24.953,C -1.5834,E1 25.0529,E2 379.5508} C_DIS
LIN {X 42.9002,Y 131.4011,Z 160,A 68.5196,B 24.953,C -1.5838,E1 25.0489,E2 378.0373} C_DIS
LIN {X 39.5361,Y 132.4517,Z 160,A 69.9828,B 24.953,C -1.5851,E1 25.045,E2 376.5737} C_DIS
LIN {X 36.2638,Y 133.3845,Z 160,A 71.4262,B 24.9528,C -1.5879,E1 25.0411,E2 375.126} C_DIS
LIN {X 32.8593,Y 134.2629,Z 160,A 72.9665,B 24.9524,C -1.5934,E1 25.0369,E2 373.575} C_DIS
LIN {X 28.4,Y 135.2779,Z 160,A 74.7261,B 24.9528,C -1.5868,E1 25.0321,E2 371.8332} C_DIS
LIN {X 24.3738,Y 136.0588,Z 160,A 76.3302,B 24.9531,C -1.5823,E1 25.0278,E2 370.2416} C_DIS
LIN {X 18.2493,Y 137.0151,Z 160,A 79.1043,B 24.9524,C -1.5942,E1 25.02,E2 367.4418} C_DIS
LIN {X 13.6776,Y 137.5472,Z 160,A 81.0487,B 24.9522,C -1.5965,E1 25.0146,E2 365.4933} C_DIS
LIN {X 9.4532,Y 137.9026,Z 160,A 82.6491,B 24.9527,C -1.5881,E1 25.0102,E2 363.9137} C_DIS
LIN {X 6.159,Y 138.0897,Z 160,A 84.042,B 24.9527,C -1.5894,E1 25.0063,E2 362.5182} C_DIS
LIN {X 2.9803,Y 138.1945,Z 160,A 85.3578,B 24.9527,C -1.5891,E1 25.0027,E2 361.2034} C_DIS
LIN {X -0.7546,Y 138.2229,Z 160,A 86.9538,B 24.9525,C -1.5915,E1 24.9982,E2 359.6018} C_DIS
LIN {X -4.2308,Y 138.1607,Z 160,A 88.3204,B 24.9528,C -1.587,E1 24.9944,E2 358.2457} C_DIS
LIN {X -9.1912,Y 137.9207,Z 160,A 90.3844,B 24.9528,C -1.5865,E1 24.9887,E2 356.1823} C_DIS
LIN {X -12.8743,Y 137.6244,Z 160,A 91.9735,B 24.9527,C -1.5889,E1 24.9842,E2 354.5867} C_DIS
LIN {X -16.3874,Y 137.2499,Z 160,A 93.4054,B 24.9529,C -1.5863,E1 24.9803,E2 353.1601} C_DIS
LIN {X -19.8804,Y 136.788,Z 160,A 94.8624,B 24.9529,C -1.5852,E1 24.9762,E2 351.7046} C_DIS
LIN {X -23.9476,Y 136.135,Z 160,A 96.4468,B 24.9534,C -1.5773,E1 24.9719,E2 350.1373} C_DIS
LIN {X -27.0007,Y 135.5631,Z 160,A 97.8771,B 24.953,C -1.5839,E1 24.9679,E2 348.6899} C_DIS
LIN {X -30.3396,Y 134.8546,Z 160,A 99.3176,B 24.953,C -1.5839,E1 24.964,E2 347.2474} C_DIS
LIN {X -33.7541,Y 134.0402,Z 160,A 100.77,B 24.953,C -1.5824,E1 24.9601,E2 345.7967} C_DIS
LIN {X -36.7913,Y 133.239,Z 160,A 102.0754,B 24.9532,C -1.5812,E1 24.9566,E2 344.4921} C_DIS
LIN {X -40.1177,Y 132.2751,Z 160,A 103.4776,B 24.9534,C -1.5778,E1 24.9528,E2 343.0957} C_DIS
LIN {X -43.3647,Y 131.2464,Z 160,A 104.921,B 24.9534,C -1.5778,E1 24.949,E2 341.6497} C_DIS
LIN {X -47.2576,Y 129.8956,Z 160,A 106.6193,B 24.9535,C -1.575,E1 24.9445,E2 339.9545} C_DIS
LIN {X -51.1049,Y 128.4316,Z 160,A 108.4392,B 24.9533,C -1.5787,E1 24.9398,E2 338.1222} C_DIS
LIN {X -54.7625,Y 126.9136,Z 160,A 109.9742,B 24.9538,C -1.5706,E1 24.9358,E2 336.6027} C_DIS
LIN {X -57.8775,Y 125.5237,Z 160,A 111.4144,B 24.9538,C -1.5698,E1 24.9322,E2 335.1608} C_DIS
LIN {X -61.9784,Y 123.5529,Z 160,A 113.2758,B 24.9541,C -1.5654,E1 24.9275,E2 333.3051} C_DIS
LIN {X -65.2011,Y 121.8828,Z 160,A 114.9141,B 24.9538,C -1.5699,E1 24.9234,E2 331.6517} C_DIS
LIN {X -68.712,Y 119.9385,Z 160,A 116.579,B 24.954,C -1.5669,E1 24.9194,E2 329.9889} C_DIS
LIN {X -72.435,Y 117.7273,Z 160,A 118.3829,B 24.9542,C -1.564,E1 24.9151,E2 328.1864} C_DIS
LIN {X -75.8239,Y 115.5738,Z 160,A 119.9571,B 24.9546,C -1.556,E1 24.9114,E2 326.6261} C_DIS
LIN {X -78.7102,Y 113.6279,Z 160,A 121.4047,B 24.9548,C -1.5533,E1 24.9081,E2 325.18} C_DIS
LIN {X -81.9959,Y 111.2799,Z 160,A 123.1121,B 24.9548,C -1.5515,E1 24.9042,E2 323.4709} C_DIS
LIN {X -85.3277,Y 108.746,Z 160,A 124.92,B 24.9548,C -1.5515,E1 24.9002,E2 321.6563} C_DIS
LIN {X -88.5725,Y 106.1205,Z 160,A 126.5423,B 24.9554,C -1.542,E1 24.8968,E2 320.0506} C_DIS
LIN {X -91.2293,Y 103.8457,Z 160,A 128.0115,B 24.9556,C -1.5397,E1 24.8937,E2 318.5812} C_DIS
LIN {X -93.7446,Y 101.5802,Z 160,A 129.4353,B 24.9557,C -1.5374,E1 24.8907,E2 317.157} C_DIS
LIN {X -96.472,Y 98.9943,Z 160,A 131.0046,B 24.9559,C -1.5342,E1 24.8876,E2 315.5889} C_DIS
LIN {X -99.4894,Y 95.9607,Z 160,A 132.7866,B 24.9561,C -1.5302,E1 24.8841,E2 313.8088} C_DIS
LIN {X -101.9667,Y 93.3242,Z 160,A 134.4213,B 24.956,C -1.5333,E1 24.881,E2 312.1595} C_DIS
LIN {X -105.1641,Y 89.7056,Z 160,A 136.3998,B 24.9563,C -1.5268,E1 24.8774,E2 310.1874} C_DIS
LIN {X -107.8566,Y 86.4503,Z 160,A 138.1983,B 24.9565,C -1.5245,E1 24.8742,E2 308.386} C_DIS
LIN {X -110.4528,Y 83.1067,Z 160,A 139.8099,B 24.9572,C -1.5123,E1 24.8715,E2 306.7958} C_DIS
LIN {X -112.4823,Y 80.3384,Z 160,A 141.2375,B 24.9574,C -1.5086,E1 24.8692,E2 305.3701} C_DIS
LIN {X -114.4428,Y 77.5201,Z 160,A 142.6676,B 24.9576,C -1.5049,E1 24.8669,E2 303.9417} C_DIS
LIN {X -116.7057,Y 74.0704,Z 160,A 144.5229,B 24.9574,C -1.5074,E1 24.8641,E2 302.0712} C_DIS
LIN {X -119.1407,Y 70.0858,Z 160,A 146.4178,B 24.9579,C -1.4996,E1 24.8614,E2 300.1851} C_DIS
LIN {X -121.0226,Y 66.784,Z 160,A 147.9416,B 24.9583,C -1.4922,E1 24.8593,E2 298.6708} C_DIS
LIN {X -122.9958,Y 63.0727,Z 160,A 149.7358,B 24.9584,C -1.4896,E1 24.857,E2 296.8733} C_DIS
LIN {X -124.653,Y 59.7297,Z 160,A 151.2371,B 24.9588,C -1.4826,E1 24.8551,E2 295.3807} C_DIS
LIN {X -126.0806,Y 56.6544,Z 160,A 152.6766,B 24.959,C -1.48,E1 24.8535,E2 293.9395} C_DIS
LIN {X -127.4744,Y 53.4443,Z 160,A 154.1369,B 24.9592,C -1.4759,E1 24.8519,E2 292.4808} C_DIS
LIN {X -128.7878,Y 50.1968,Z 160,A 155.5756,B 24.9595,C -1.4706,E1 24.8504,E2 291.0466} C_DIS
LIN {X -129.9834,Y 47.0141,Z 160,A 156.7904,B 24.9603,C -1.4562,E1 24.8492,E2 289.8592} C_DIS
LIN {X -131.0212,Y 44.0411,Z 160,A 158.3088,B 24.9599,C -1.4629,E1 24.8478,E2 288.3163} C_DIS
LIN {X -132.0935,Y 40.7112,Z 160,A 159.768,B 24.9601,C -1.4587,E1 24.8466,E2 286.8588} C_DIS
LIN {X -133.0492,Y 37.4699,Z 160,A 161.2019,B 24.9603,C -1.4559,E1 24.8455,E2 285.4233} C_DIS
LIN {X -133.9784,Y 33.9976,Z 160,A 162.6761,B 24.9606,C -1.4502,E1 24.8445,E2 283.954} C_DIS
LIN {X -134.7667,Y 30.7243,Z 160,A 164.0819,B 24.9608,C -1.4461,E1 24.8436,E2 282.5496} C_DIS
LIN {X -135.3496,Y 28.0499,Z 160,A 165.2327,B 24.961,C -1.4432,E1 24.8429,E2 281.3991} C_DIS
LIN {X -136.0373,Y 24.4934,Z 160,A 166.7391,B 24.9612,C -1.4385,E1 24.8422,E2 279.8949} C_DIS
LIN {X -136.5969,Y 21.1507,Z 160,A 168.1706,B 24.9614,C -1.4352,E1 24.8415,E2 278.4627} C_DIS
LIN {X -137.0908,Y 17.6712,Z 160,A 169.6242,B 24.9617,C -1.4302,E1 24.841,E2 277.0124} C_DIS
LIN {X -137.4962,Y 14.1864,Z 160,A 171.1384,B 24.9617,C -1.4284,E1 24.8405,E2 275.4933} C_DIS
LIN {X -137.8249,Y 10.5176,Z 160,A 172.6797,B 24.962,C -1.4241,E1 24.8402,E2 273.9531} C_DIS
LIN {X -138.0475,Y 7.0012,Z 160,A 174.0962,B 24.9624,C -1.417,E1 24.8399,E2 272.545} C_DIS
LIN {X -138.1817,Y 3.4746,Z 160,A 175.5524,B 24.9627,C -1.4118,E1 24.8399,E2 271.0924} C_DIS
LIN {X -138.228,Y 0.0624,Z 160,A 177.1052,B 24.9625,C -1.4142,E1 24.8398,E2 269.5247} C_DIS
LIN {X -138.1561,Y -4.3974,Z 160,A 178.8565,B 24.9631,C -1.4031,E1 24.8399,E2 267.7893} C_DIS
LIN {X -137.9922,Y -8.0296,Z 160,A -179.6143,B 24.9633,C -1.3992,E1 24.8401,E2 266.26} C_DIS
LIN {X -137.7511,Y -11.4355,Z 160,A -178.1767,B 24.9635,C -1.3957,E1 24.8404,E2 264.8222} C_DIS
LIN {X -137.4067,Y -15.0186,Z 160,A -176.6851,B 24.9638,C -1.3908,E1 24.8409,E2 263.3333} C_DIS
LIN {X -136.9689,Y -18.6015,Z 160,A -175.2074,B 24.9641,C -1.385,E1 24.8414,E2 261.8607} C_DIS
LIN {X -136.4518,Y -22.0779,Z 160,A -173.717,B 24.9642,C -1.3819,E1 24.842,E2 260.3686} C_DIS
LIN {X -135.7974,Y -25.7907,Z 160,A -172.153,B 24.9645,C -1.377,E1 24.8428,E2 258.8071} C_DIS
LIN {X -135.126,Y -29.1037,Z 160,A -170.7446,B 24.9647,C -1.3729,E1 24.8436,E2 257.4002} C_DIS
LIN {X -134.3732,Y -32.402,Z 160,A -169.318,B 24.9649,C -1.3697,E1 24.8445,E2 255.973} C_DIS
LIN {X -133.2863,Y -36.6221,Z 160,A -167.2693,B 24.9645,C -1.3764,E1 24.846,E2 253.8962} C_DIS
LIN {X -131.5503,Y -42.4344,Z 160,A -164.9707,B 24.9655,C -1.3575,E1 24.8479,E2 251.6294} C_DIS
LIN {X -130.182,Y -46.4633,Z 160,A -163.3073,B 24.966,C -1.3469,E1 24.8494,E2 249.9818} C_DIS
LIN {X -129.1042,Y -49.3828,Z 160,A -161.9082,B 24.966,C -1.3486,E1 24.8508,E2 248.5707} C_DIS
LIN {X -127.7244,Y -52.8457,Z 160,A -160.4206,B 24.9663,C -1.341,E1 24.8523,E2 247.093} C_DIS
LIN {X -126.3056,Y -56.1514,Z 160,A -158.8222,B 24.9663,C -1.3422,E1 24.8541,E2 245.4831} C_DIS
LIN {X -124.8459,Y -59.326,Z 160,A -157.3837,B 24.9665,C -1.3375,E1 24.8558,E2 244.0479} C_DIS
LIN {X -123.3493,Y -62.3784,Z 160,A -155.9697,B 24.9667,C -1.3337,E1 24.8576,E2 242.6354} C_DIS
LIN {X -121.7885,Y -65.3765,Z 160,A -154.4427,B 24.9666,C -1.3362,E1 24.8596,E2 241.0942} C_DIS
LIN {X -119.6214,Y -69.2622,Z 160,A -152.692,B 24.9671,C -1.3262,E1 24.862,E2 239.3581} C_DIS
LIN {X -117.8169,Y -72.289,Z 160,A -151.2428,B 24.9673,C -1.3216,E1 24.8641,E2 237.9124} C_DIS
LIN {X -115.783,Y -75.5043,Z 160,A -149.6481,B 24.9674,C -1.3183,E1 24.8665,E2 236.3175} C_DIS
LIN {X -113.4948,Y -78.9016,Z 160,A -147.8764,B 24.9674,C -1.3178,E1 24.8693,E2 234.5383} C_DIS
LIN {X -111.4073,Y -81.8225,Z 160,A -146.4157,B 24.9677,C -1.3125,E1 24.8717,E2 233.083} C_DIS
LIN {X -109.2225,Y -84.717,Z 160,A -144.9434,B 24.968,C -1.3071,E1 24.8742,E2 231.6165} C_DIS
LIN {X -107.0331,Y -87.4668,Z 160,A -143.4201,B 24.968,C -1.3071,E1 24.8769,E2 230.0863} C_DIS
LIN {X -104.1462,Y -90.885,Z 160,A -141.6079,B 24.9683,C -1.3004,E1 24.8801,E2 228.2816} C_DIS
LIN {X -101.3796,Y -93.9617,Z 160,A -139.8333,B 24.9683,C -1.2996,E1 24.8835,E2 226.5011} C_DIS
LIN {X -98.6503,Y -96.8227,Z 160,A -138.1154,B 24.9683,C -1.3001,E1 24.8869,E2 224.7746} C_DIS
LIN {X -95.3589,Y -100.0662,Z 160,A -136.2229,B 24.9686,C -1.2948,E1 24.8906,E2 222.887} C_DIS
LIN {X -92.0259,Y -103.1398,Z 160,A -134.2915,B 24.9686,C -1.2937,E1 24.8946,E2 220.9504} C_DIS
LIN {X -88.8587,Y -105.8803,Z 160,A -132.5703,B 24.9689,C -1.2894,E1 24.8983,E2 219.2326} C_DIS
LIN {X -85.2775,Y -108.7855,Z 160,A -130.6915,B 24.9691,C -1.2841,E1 24.9024,E2 217.3596} C_DIS
LIN {X -82.0897,Y -111.211,Z 160,A -129.1074,B 24.9695,C -1.277,E1 24.9059,E2 215.7865} C_DIS
LIN {X -79.2275,Y -113.268,Z 160,A -127.5393,B 24.9693,C -1.2802,E1 24.9095,E2 214.2056} C_DIS
LIN {X -75.6386,Y -115.6958,Z 160,A -125.7187,B 24.9693,C -1.2785,E1 24.9138,E2 212.3829} C_DIS
LIN {X -71.8652,Y -118.0766,Z 160,A -123.9595,B 24.9698,C -1.2709,E1 24.9179,E2 210.6364} C_DIS
LIN {X -68.7765,Y -119.9017,Z 160,A -122.4961,B 24.9699,C -1.2674,E1 24.9214,E2 209.1768} C_DIS
LIN {X -65.2151,Y -121.8752,Z 160,A -120.7237,B 24.9699,C -1.2696,E1 24.9258,E2 207.3942} C_DIS
LIN {X -61.759,Y -123.6619,Z 160,A -119.1781,B 24.9701,C -1.2639,E1 24.9296,E2 205.858} C_DIS
LIN {X -58.5772,Y -125.2002,Z 160,A -117.7116,B 24.9701,C -1.2622,E1 24.9333,E2 204.3917} C_DIS
LIN {X -54.9571,Y -126.8295,Z 160,A -115.9767,B 24.9701,C -1.2652,E1 24.9378,E2 202.6457} C_DIS
LIN {X -51.1665,Y -128.4067,Z 160,A -114.2115,B 24.9699,C -1.2668,E1 24.9424,E2 200.8726} C_DIS
LIN {X -47.1228,Y -129.9443,Z 160,A -112.5317,B 24.9703,C -1.259,E1 24.9467,E2 199.2079} C_DIS
LIN {X -43.7978,Y -131.1022,Z 160,A -111.0937,B 24.9704,C -1.2566,E1 24.9505,E2 197.7729} C_DIS
LIN {X -39.5809,Y -132.4385,Z 160,A -109.2547,B 24.9704,C -1.2555,E1 24.9554,E2 195.9334} C_DIS
LIN {X -36.3039,Y -133.3738,Z 160,A -107.8038,B 24.9704,C -1.2566,E1 24.9593,E2 194.4775} C_DIS
LIN {X -32.7593,Y -134.287,Z 160,A -106.2262,B 24.9704,C -1.2591,E1 24.9636,E2 192.8918} C_DIS
LIN {X -28.5357,Y -135.2486,Z 160,A -104.537,B 24.9706,C -1.2523,E1 24.9682,E2 191.2164} C_DIS
LIN {X -25.1791,Y -135.9143,Z 160,A -103.1208,B 24.9706,C -1.2516,E1 24.9721,E2 189.8004} C_DIS
LIN {X -21.9552,Y -136.4722,Z 160,A -101.7672,B 24.9706,C -1.2511,E1 24.9758,E2 188.4469} C_DIS
LIN {X -18.243,Y -137.0159,Z 160,A -100.0851,B 24.9704,C -1.2577,E1 24.9805,E2 186.7477} C_DIS
LIN {X -14.1282,Y -137.5025,Z 160,A -98.4953,B 24.9707,C -1.2504,E1 24.9849,E2 185.1741} C_DIS
LIN {X -10.7091,Y -137.8109,Z 160,A -97.0519,B 24.9707,C -1.2515,E1 24.9889,E2 183.7275} C_DIS
LIN {X -6.6564,Y -138.0648,Z 160,A -95.3148,B 24.9705,C -1.2546,E1 24.9938,E2 181.9827} C_DIS
LIN {X -2.5056,Y -138.2024,Z 160,A -93.6499,B 24.9707,C -1.2517,E1 24.9984,E2 180.3244} C_DIS
LIN {X 0.9745,Y -138.2214,Z 160,A -92.2368,B 24.9707,C -1.2504,E1 25.0023,E2 178.9144} C_DIS
Enddeposition()
LIN {X 0.9745,Y -138.2214,Z 160,A -92.2368,B 24.9707,C -1.2504,E1 25.0023,E2 178.9144} C_DIS
Startdeposition()
$VEL.CP = VEL_PRINT
LIN {X -1.1068,Y -137.295,Z 160,A -94.2449,B 24.9728,C -1.2043,E1 24.9964,E2 181.0316} C_DIS
LIN {X -5.5524,Y -137.1868,Z 160,A -95.6149,B 24.9717,C -1.2303,E1 24.9928,E2 182.3403} C_DIS
LIN {X -9.75,Y -136.9525,Z 160,A -97.316,B 24.9715,C -1.2331,E1 24.9881,E2 184.0353} C_DIS
LIN {X -13.5104,Y -136.6331,Z 160,A -98.9189,B 24.9715,C -1.2317,E1 24.9836,E2 185.6423} C_DIS
LIN {X -18.7861,Y -136.0091,Z 160,A -101.2807,B 24.9719,C -1.2243,E1 24.977,E2 188.0233} C_DIS
LIN {X -26.0291,Y -134.8091,Z 160,A -104.5513,B 24.9724,C -1.2144,E1 24.9679,E2 191.3209} C_DIS
LIN {X -29.6496,Y -134.0609,Z 160,A -105.8657,B 24.9718,C -1.2272,E1 24.9644,E2 192.6063} C_DIS
LIN {X -33.6237,Y -133.118,Z 160,A -107.5115,B 24.9716,C -1.2314,E1 24.96,E2 194.2446} C_DIS
LIN {X -37.726,Y -132.0162,Z 160,A -109.3769,B 24.9718,C -1.2276,E1 24.9549,E2 196.122} C_DIS
LIN {X -41.5811,Y -130.8509,Z 160,A -110.9466,B 24.9714,C -1.2348,E1 24.9508,E2 197.6774} C_DIS
LIN {X -44.9071,Y -129.7469,Z 160,A -112.3637,B 24.9713,C -1.2384,E1 24.947,E2 199.0884} C_DIS
LIN {X -49.1434,Y -128.2039,Z 160,A -114.3457,B 24.9714,C -1.2348,E1 24.9418,E2 201.083} C_DIS
LIN {X -52.5245,Y -126.8552,Z 160,A -115.6241,B 24.9708,C -1.2492,E1 24.9386,E2 202.3302} C_DIS
LIN {X -56.3399,Y -125.2069,Z 160,A -117.5659,B 24.9712,C -1.2401,E1 24.9336,E2 204.2981} C_DIS
LIN {X -60.3925,Y -123.3035,Z 160,A -119.4311,B 24.9711,C -1.2426,E1 24.9289,E2 206.1622} C_DIS
LIN {X -63.4114,Y -121.7788,Z 160,A -120.8375,B 24.971,C -1.2447,E1 24.9254,E2 207.5674} C_DIS
LIN {X -66.6822,Y -120.0205,Z 160,A -122.452,B 24.971,C -1.2434,E1 24.9214,E2 209.1895} C_DIS
LIN {X -70.4624,Y -117.841,Z 160,A -124.0954,B 24.9705,C -1.2554,E1 24.9175,E2 210.8094} C_DIS
LIN {X -73.821,Y -115.7667,Z 160,A -125.9631,B 24.9709,C -1.2465,E1 24.913,E2 212.7042} C_DIS
LIN {X -77.7018,Y -113.1982,Z 160,A -127.8438,B 24.9706,C -1.2529,E1 24.9087,E2 214.5759} C_DIS
LIN {X -81.0272,Y -110.8427,Z 160,A -129.5787,B 24.9706,C -1.2541,E1 24.9047,E2 216.314} C_DIS
LIN {X -84.6987,Y -108.0627,Z 160,A -131.5265,B 24.9704,C -1.2563,E1 24.9004,E2 218.2637} C_DIS
LIN {X -91.9164,Y -101.9949,Z 160,A -135.4935,B 24.9702,C -1.2624,E1 24.892,E2 222.2315} C_DIS
LIN {X -95.2544,Y -98.8843,Z 160,A -137.3288,B 24.9698,C -1.27,E1 24.8883,E2 224.0564} C_DIS
LIN {X -98.4318,Y -95.7219,Z 160,A -139.2782,B 24.9698,C -1.27,E1 24.8844,E2 226.014} C_DIS
LIN {X -100.7507,Y -93.2784,Z 160,A -140.7161,B 24.9698,C -1.2716,E1 24.8817,E2 227.4544} C_DIS
LIN {X -102.927,Y -90.8704,Z 160,A -142.2397,B 24.97,C -1.2661,E1 24.8788,E2 228.998} C_DIS
LIN {X -105.0683,Y -88.3861,Z 160,A -143.4055,B 24.9693,C -1.2797,E1 24.8768,E2 230.1367} C_DIS
LIN {X -107.7988,Y -85.0348,Z 160,A -145.2478,B 24.9693,C -1.2822,E1 24.8736,E2 231.9818} C_DIS
LIN {X -110.4037,Y -81.6248,Z 160,A -147.0723,B 24.9691,C -1.285,E1 24.8705,E2 233.8084} C_DIS
LIN {X -112.9599,Y -78.0478,Z 160,A -149.5942,B 24.9705,C -1.255,E1 24.8664,E2 236.414} C_DIS
LIN {X -116.3091,Y -72.964,Z 160,A -151.4535,B 24.9685,C -1.2961,E1 24.8637,E2 238.1848} C_DIS
LIN {X -118.6099,Y -69.1613,Z 160,A -153.3199,B 24.9683,C -1.3006,E1 24.861,E2 240.0503} C_DIS
LIN {X -120.9038,Y -65.0669,Z 160,A -155.3611,B 24.9683,C -1.3019,E1 24.8583,E2 242.0991} C_DIS
LIN {X -123.0032,Y -61.0013,Z 160,A -157.8436,B 24.9694,C -1.2787,E1 24.8551,E2 244.6502} C_DIS
LIN {X -125.4399,Y -55.8192,Z 160,A -159.5098,B 24.9673,C -1.322,E1 24.8533,E2 246.2225} C_DIS
LIN {X -126.9639,Y -52.2642,Z 160,A -161.2462,B 24.9673,C -1.3206,E1 24.8514,E2 247.9719} C_DIS
LIN {X -128.4093,Y -48.602,Z 160,A -162.8121,B 24.9669,C -1.3294,E1 24.8498,E2 249.5255} C_DIS
LIN {X -129.6399,Y -45.2157,Z 160,A -164.2997,B 24.9666,C -1.3348,E1 24.8484,E2 251.0087} C_DIS
LIN {X -130.7262,Y -41.9715,Z 160,A -165.7824,B 24.9666,C -1.3365,E1 24.8472,E2 252.4959} C_DIS
LIN {X -131.9526,Y -37.9454,Z 160,A -167.7243,B 24.9667,C -1.3326,E1 24.8456,E2 254.4582} C_DIS
LIN {X -133.175,Y -33.3991,Z 160,A -169.5994,B 24.9662,C -1.3433,E1 24.8443,E2 256.3187} C_DIS
LIN {X -134.1612,Y -29.185,Z 160,A -171.1702,B 24.9653,C -1.3609,E1 24.8433,E2 257.8569} C_DIS
LIN {X -135.0751,Y -24.6143,Z 160,A -173.2681,B 24.9653,C -1.3594,E1 24.8422,E2 259.9707} C_DIS
LIN {X -135.6665,Y -21.1086,Z 160,A -174.7565,B 24.9652,C -1.364,E1 24.8416,E2 261.457} C_DIS
LIN {X -136.192,Y -17.4039,Z 160,A -176.4203,B 24.9652,C -1.364,E1 24.8409,E2 263.1309} C_DIS
LIN {X -136.6652,Y -13.176,Z 160,A -178.102,B 24.9646,C -1.3745,E1 24.8404,E2 264.7976} C_DIS
LIN {X -136.9861,Y -9.2902,Z 160,A -179.8716,B 24.9647,C -1.3727,E1 24.8401,E2 266.5821} C_DIS
LIN {X -137.1981,Y -5.2622,Z 160,A 178.5312,B 24.9642,C -1.3826,E1 24.8399,E2 268.1653} C_DIS
LIN {X -137.2964,Y -0.9581,Z 160,A 176.8379,B 24.9636,C -1.3937,E1 24.8398,E2 269.8424} C_DIS
LIN {X -137.2779,Y 2.4109,Z 160,A 175.2913,B 24.9637,C -1.3913,E1 24.8398,E2 271.4039} C_DIS
LIN {X -137.146,Y 6.4923,Z 160,A 173.5768,B 24.9635,C -1.3964,E1 24.84,E2 273.1166} C_DIS
LIN {X -136.9307,Y 10.0488,Z 160,A 172.107,B 24.9632,C -1.4023,E1 24.8403,E2 274.5813} C_DIS
LIN {X -136.5531,Y 14.2965,Z 160,A 170.323,B 24.9629,C -1.4079,E1 24.8408,E2 276.3626} C_DIS
LIN {X -136.1312,Y 17.8684,Z 160,A 168.8196,B 24.9626,C -1.4128,E1 24.8413,E2 277.8633} C_DIS
LIN {X -135.5958,Y 21.5652,Z 160,A 167.143,B 24.9626,C -1.4121,E1 24.842,E2 279.5517} C_DIS
LIN {X -134.891,Y 25.6007,Z 160,A 165.5356,B 24.9621,C -1.4228,E1 24.8428,E2 281.143} C_DIS
LIN {X -134.2292,Y 28.8698,Z 160,A 164.0934,B 24.962,C -1.4249,E1 24.8436,E2 282.5887} C_DIS
LIN {X -133.3985,Y 32.4942,Z 160,A 162.5461,B 24.9617,C -1.4302,E1 24.8446,E2 284.1325} C_DIS
LIN {X -132.4305,Y 36.2442,Z 160,A 160.8644,B 24.9616,C -1.4321,E1 24.8458,E2 285.8193} C_DIS
LIN {X -131.5182,Y 39.427,Z 160,A 159.4469,B 24.9614,C -1.4348,E1 24.8469,E2 287.2386} C_DIS
LIN {X -130.0179,Y 44.1232,Z 160,A 157.3647,B 24.9611,C -1.4402,E1 24.8487,E2 289.3199} C_DIS
LIN {X -128.6982,Y 47.8308,Z 160,A 155.8171,B 24.9606,C -1.4502,E1 24.8502,E2 290.8524} C_DIS
LIN {X -127.4286,Y 51.1165,Z 160,A 154.342,B 24.9604,C -1.4546,E1 24.8517,E2 292.3254} C_DIS
LIN {X -126.2208,Y 54.0317,Z 160,A 152.977,B 24.9603,C -1.4563,E1 24.8532,E2 293.6939} C_DIS
LIN {X -124.8362,Y 57.1581,Z 160,A 151.5407,B 24.9601,C -1.4603,E1 24.8548,E2 295.1286} C_DIS
LIN {X -123.3264,Y 60.3461,Z 160,A 150.0088,B 24.96,C -1.4618,E1 24.8567,E2 296.6651} C_DIS
LIN {X -121.7727,Y 63.4231,Z 160,A 148.6547,B 24.9595,C -1.4704,E1 24.8584,E2 298.006} C_DIS
LIN {X -119.0536,Y 68.3946,Z 160,A 146.1441,B 24.9595,C -1.4701,E1 24.8618,E2 300.5304} C_DIS
LIN {X -116.6966,Y 72.342,Z 160,A 144.0694,B 24.9596,C -1.468,E1 24.8649,E2 302.6208} C_DIS
LIN {X -113.9331,Y 76.6212,Z 160,A 142.1272,B 24.9588,C -1.4833,E1 24.8678,E2 304.5364} C_DIS
LIN {X -111.6704,Y 79.8819,Z 160,A 140.4979,B 24.9584,C -1.4893,E1 24.8704,E2 306.1593} C_DIS
LIN {X -109.3544,Y 83.0251,Z 160,A 138.7842,B 24.9584,C -1.4896,E1 24.8733,E2 307.8806} C_DIS
LIN {X -106.1245,Y 87.1154,Z 160,A 136.4129,B 24.9587,C -1.4856,E1 24.8775,E2 310.2723} C_DIS
LIN {X -104.0192,Y 89.6182,Z 160,A 135.236,B 24.9579,C -1.4987,E1 24.8796,E2 311.4236} C_DIS
LIN {X -101.0448,Y 92.9588,Z 160,A 133.4147,B 24.9575,C -1.5058,E1 24.883,E2 313.236} C_DIS
LIN {X -98.2854,Y 95.8724,Z 160,A 131.6444,B 24.9575,C -1.5052,E1 24.8864,E2 315.0154} C_DIS
LIN {X -95.0409,Y 99.0893,Z 160,A 129.7589,B 24.9572,C -1.511,E1 24.8902,E2 316.8951} C_DIS
LIN {X -91.7885,Y 102.1094,Z 160,A 127.902,B 24.957,C -1.5151,E1 24.894,E2 318.7495} C_DIS
LIN {X -88.4135,Y 105.0453,Z 160,A 126.0131,B 24.9568,C -1.5183,E1 24.898,E2 320.6382} C_DIS
LIN {X -86.0473,Y 106.992,Z 160,A 124.6193,B 24.957,C -1.5153,E1 24.9011,E2 322.0443} C_DIS
LIN {X -81.8798,Y 110.214,Z 160,A 122.6204,B 24.9561,C -1.5302,E1 24.9055,E2 324.015} C_DIS
LIN {X -79.0077,Y 112.2907,Z 160,A 121.1191,B 24.9561,C -1.5322,E1 24.9089,E2 325.5169} C_DIS
LIN {X -75.6348,Y 114.5897,Z 160,A 119.528,B 24.9555,C -1.5413,E1 24.9125,E2 327.0915} C_DIS
LIN {X -73.369,Y 116.0535,Z 160,A 118.1291,B 24.9562,C -1.5296,E1 24.9159,E2 328.5229} C_DIS
LIN {X -70.0761,Y 118.0713,Z 160,A 115.6118,B 24.9586,C -1.4867,E1 24.9223,E2 331.1496} C_DIS
LIN {X -63.6211,Y 121.6687,Z 160,A 113.6577,B 24.955,C -1.5495,E1 24.9267,E2 332.9601} C_DIS
LIN {X -61.3227,Y 122.8446,Z 160,A 112.39,B 24.9555,C -1.5414,E1 24.9299,E2 334.2502} C_DIS
LIN {X -58.057,Y 124.4206,Z 160,A 110.9385,B 24.9552,C -1.547,E1 24.9335,E2 335.6921} C_DIS
LIN {X -54.7201,Y 125.9232,Z 160,A 109.4893,B 24.9548,C -1.5534,E1 24.9372,E2 337.1297} C_DIS
LIN {X -52.0943,Y 127.0344,Z 160,A 107.7935,B 24.9562,C -1.529,E1 24.9418,E2 338.8871} C_DIS
LIN {X -48.2977,Y 128.5233,Z 160,A 106.5723,B 24.9546,C -1.5561,E1 24.9448,E2 340.0466} C_DIS
LIN {X -45.2569,Y 129.6256,Z 160,A 105.2626,B 24.9544,C -1.56,E1 24.9482,E2 341.3497} C_DIS
LIN {X -41.7029,Y 130.812,Z 160,A 103.8376,B 24.9539,C -1.5691,E1 24.9519,E2 342.7558} C_DIS
LIN {X -35.864,Y 132.5328,Z 160,A 101.0827,B 24.9544,C -1.5607,E1 24.9594,E2 345.5351} C_DIS
LIN {X -32.3615,Y 133.4305,Z 160,A 99.5715,B 24.9543,C -1.562,E1 24.9635,E2 347.0452} C_DIS
LIN {X -28.7221,Y 134.2611,Z 160,A 97.9699,B 24.9543,C -1.5612,E1 24.9678,E2 348.6509} C_DIS
LIN {X -24.4683,Y 135.1012,Z 160,A 96.1974,B 24.9541,C -1.5646,E1 24.9727,E2 350.4172} C_DIS
LIN {X -21.0972,Y 135.6683,Z 160,A 94.8071,B 24.954,C -1.5675,E1 24.9765,E2 351.8018} C_DIS
LIN {X -17.5612,Y 136.1714,Z 160,A 93.1885,B 24.9543,C -1.5617,E1 24.981,E2 353.4354} C_DIS
LIN {X -13.4072,Y 136.643,Z 160,A 91.4687,B 24.9542,C -1.564,E1 24.9858,E2 355.1509} C_DIS
LIN {X -9.2031,Y 136.9922,Z 160,A 89.8115,B 24.9538,C -1.5702,E1 24.9904,E2 356.7941} C_DIS
LIN {X -3.7614,Y 137.2475,Z 160,A 86.6942,B 24.9563,C -1.5266,E1 24.9994,E2 360.0151} C_DIS
LIN {X 2.2836,Y 137.28,Z 160,A 85.1435,B 24.9533,C -1.5782,E1 25.0034,E2 361.4433} C_DIS
LIN {X 9.4456,Y 136.9748,Z 160,A 81.2829,B 24.956,C -1.5322,E1 25.0144,E2 365.4115} C_DIS
LIN {X 14.8563,Y 136.4929,Z 160,A 79.6959,B 24.9539,C -1.568,E1 25.0186,E2 366.9129} C_DIS
LIN {X 17.7134,Y 136.1515,Z 160,A 78.367,B 24.9544,C -1.5608,E1 25.0223,E2 368.2577} C_DIS
LIN {X 23.252,Y 135.3172,Z 160,A 75.8594,B 24.9549,C -1.551,E1 25.0293,E2 370.7861} C_DIS
LIN {X 26.6607,Y 134.6874,Z 160,A 74.6217,B 24.9543,C -1.5615,E1 25.0326,E2 371.9975} C_DIS
LIN {X 30.4022,Y 133.8905,Z 160,A 73.2063,B 24.9538,C -1.5704,E1 25.0364,E2 373.3899} C_DIS
LIN {X 33.6081,Y 133.122,Z 160,A 71.7735,B 24.954,C -1.5665,E1 25.0403,E2 374.8298} C_DIS
LIN {X 36.8205,Y 132.2694,Z 160,A 70.3404,B 24.9542,C -1.5631,E1 25.0442,E2 376.2687} C_DIS
LIN {X 40.139,Y 131.3003,Z 160,A 68.9289,B 24.9542,C -1.5637,E1 25.0479,E2 377.6764} C_DIS
LIN {X 43.3568,Y 130.2731,Z 160,A 67.4676,B 24.9544,C -1.5597,E1 25.0518,E2 379.1444} C_DIS
LIN {X 47.5536,Y 128.802,Z 160,A 65.5943,B 24.9546,C -1.557,E1 25.0568,E2 381.0202} C_DIS
LIN {X 50.4631,Y 127.6908,Z 160,A 64.1188,B 24.9552,C -1.5461,E1 25.0607,E2 382.5182} C_DIS
LIN {X 55.2737,Y 125.6837,Z 160,A 62.09,B 24.9549,C -1.5516,E1 25.0658,E2 384.5291} C_DIS
LIN {X 58.9079,Y 124.0194,Z 160,A 60.6083,B 24.9544,C -1.5597,E1 25.0695,E2 385.9877} C_DIS
LIN {X 61.8929,Y 122.5575,Z 160,A 59.1232,B 24.9548,C -1.5526,E1 25.0733,E2 387.4858} C_DIS
LIN {X 65.3131,Y 120.7715,Z 160,A 57.4621,B 24.9551,C -1.5475,E1 25.0774,E2 389.1542} C_DIS
LIN {X 69.202,Y 118.586,Z 160,A 55.5814,B 24.9554,C -1.5437,E1 25.0819,E2 391.0382} C_DIS
LIN {X 72.2007,Y 116.7841,Z 160,A 54.0313,B 24.9558,C -1.5365,E1 25.0857,E2 392.6005} C_DIS
LIN {X 76.5271,Y 113.9962,Z 160,A 51.9929,B 24.9556,C -1.5389,E1 25.0904,E2 394.6264} C_DIS
LIN {X 79.6657,Y 111.8251,Z 160,A 50.4232,B 24.9557,C -1.5374,E1 25.094,E2 396.1942} C_DIS
LIN {X 83.0971,Y 109.2998,Z 160,A 48.675,B 24.9558,C -1.5358,E1 25.0979,E2 397.9399} C_DIS
LIN {X 86.8162,Y 106.369,Z 160,A 46.3641,B 24.9571,C -1.5135,E1 25.103,E2 400.2947} C_DIS
LIN {X 89.8955,Y 103.7803,Z 160,A 44.993,B 24.9563,C -1.5271,E1 25.1058,E2 401.6283} C_DIS
LIN {X 93.1611,Y 100.8589,Z 160,A 43.2237,B 24.9563,C -1.5266,E1 25.1095,E2 403.3918} C_DIS
LIN {X 96.3672,Y 97.8002,Z 160,A 41.3385,B 24.9567,C -1.5206,E1 25.1132,E2 405.2833} C_DIS
LIN {X 99.611,Y 94.4944,Z 160,A 39.3958,B 24.957,C -1.5157,E1 25.117,E2 407.2291} C_DIS
LIN {X 102.0745,Y 91.8275,Z 160,A 37.9105,B 24.957,C -1.5138,E1 25.1198,E2 408.7123} C_DIS
LIN {X 105.0763,Y 88.3765,Z 160,A 36.0116,B 24.9573,C -1.5098,E1 25.1233,E2 410.6121} C_DIS
LIN {X 107.5323,Y 85.3712,Z 160,A 34.4006,B 24.9575,C -1.5063,E1 25.1261,E2 412.2238} C_DIS
LIN {X 110.3805,Y 81.6561,Z 160,A 32.4998,B 24.9576,C -1.5043,E1 25.1293,E2 414.1203} C_DIS
LIN {X 112.4989,Y 78.7117,Z 160,A 30.5689,B 24.9591,C -1.477,E1 25.1325,E2 416.1061} C_DIS
LIN {X 114.9533,Y 75.0819,Z 160,A 29.114,B 24.9582,C -1.4931,E1 25.1346,E2 417.5158} C_DIS
LIN {X 117.3956,Y 71.202,Z 160,A 27.2391,B 24.9584,C -1.4901,E1 25.1374,E2 419.3884} C_DIS
LIN {X 119.3768,Y 67.828,Z 160,A 25.6254,B 24.9586,C -1.4866,E1 25.1396,E2 421.0019} C_DIS
LIN {X 121.401,Y 64.1309,Z 160,A 24.0844,B 24.9582,C -1.494,E1 25.1416,E2 422.5173} C_DIS
LIN {X 122.9321,Y 61.1454,Z 160,A 22.4773,B 24.9591,C -1.4782,E1 25.1437,E2 424.153} C_DIS
LIN {X 124.4923,Y 57.902,Z 160,A 21.1504,B 24.9588,C -1.4838,E1 25.1453,E2 425.4597} C_DIS
LIN {X 125.9389,Y 54.6837,Z 160,A 19.6673,B 24.959,C -1.4788,E1 25.1469,E2 426.9464} C_DIS
LIN {X 126.9614,Y 52.2701,Z 160,A 18.5056,B 24.9594,C -1.4717,E1 25.1482,E2 428.1185} C_DIS
LIN {X 128.4164,Y 48.5831,Z 160,A 16.8306,B 24.9598,C -1.4655,E1 25.1499,E2 429.7988} C_DIS
LIN {X 129.6272,Y 45.2523,Z 160,A 15.4408,B 24.9598,C -1.4661,E1 25.1512,E2 431.1795} C_DIS
LIN {X 131.5981,Y 39.1564,Z 160,A 12.7426,B 24.9603,C -1.4563,E1 25.1535,E2 433.8853} C_DIS
LIN {X 132.5957,Y 35.6282,Z 160,A 11.2365,B 24.9605,C -1.4529,E1 25.1546,E2 435.3909} C_DIS
LIN {X 133.4932,Y 32.1014,Z 160,A 9.7507,B 24.9606,C -1.45,E1 25.1556,E2 436.875} C_DIS
LIN {X 134.2363,Y 28.8371,Z 160,A 8.3438,B 24.9609,C -1.4449,E1 25.1564,E2 438.2857} C_DIS
LIN {X 135.0042,Y 25.0088,Z 160,A 6.6619,B 24.9613,C -1.4366,E1 25.1573,E2 439.9772} C_DIS
LIN {X 135.6598,Y 21.1521,Z 160,A 5.0817,B 24.9615,C -1.4344,E1 25.158,E2 441.5535} C_DIS
LIN {X 136.1786,Y 17.5065,Z 160,A 3.4986,B 24.9619,C -1.4267,E1 25.1586,E2 443.1454} C_DIS
LIN {X 136.5356,Y 14.4588,Z 160,A 2.0114,B 24.9627,C -1.4107,E1 25.1591,E2 444.6615} C_DIS
LIN {X 136.8505,Y 11.0976,Z 160,A 0.2311,B 24.9641,C -1.3849,E1 25.1595,E2 446.4919} C_DIS
LIN {X 137.1803,Y 5.7192,Z 160,A -1.3648,B 24.9625,C -1.4146,E1 25.1597,E2 448.0084} C_DIS
LIN {X 137.2813,Y -2.207,Z 160,A -5.2857,B 24.9649,C -1.3687,E1 25.1597,E2 452.014} C_DIS
LIN {X 137.0854,Y -7.6912,Z 160,A -6.998,B 24.9636,C -1.3939,E1 25.1595,E2 453.6567} C_DIS
LIN {X 136.6975,Y -12.8404,Z 160,A -9.0248,B 24.9636,C -1.3941,E1 25.159,E2 455.6711} C_DIS
LIN {X 136.2265,Y -17.1385,Z 160,A -11.2032,B 24.965,C -1.3667,E1 25.1583,E2 457.9012} C_DIS
LIN {X 135.7114,Y -20.8184,Z 160,A -12.3835,B 24.9642,C -1.3828,E1 25.1578,E2 459.0367} C_DIS
LIN {X 135.082,Y -24.5757,Z 160,A -14.0063,B 24.9646,C -1.3756,E1 25.157,E2 460.667} C_DIS
LIN {X 134.257,Y -28.7412,Z 160,A -15.7125,B 24.9646,C -1.3735,E1 25.1561,E2 462.3681} C_DIS
LIN {X 133.4161,Y -32.4213,Z 160,A -17.2998,B 24.965,C -1.3677,E1 25.155,E2 463.96} C_DIS
LIN {X 132.3994,Y -36.3558,Z 160,A -19.0333,B 24.9654,C -1.3599,E1 25.1538,E2 465.7017} C_DIS
LIN {X 131.3653,Y -39.9267,Z 160,A -20.6239,B 24.9657,C -1.3527,E1 25.1525,E2 467.3004} C_DIS
LIN {X 129.9008,Y -44.4633,Z 160,A -22.5594,B 24.9659,C -1.3493,E1 25.1508,E2 469.2327} C_DIS
LIN {X 128.6452,Y -47.9724,Z 160,A -24.0462,B 24.9659,C -1.3483,E1 25.1494,E2 470.7137} C_DIS
LIN {X 126.913,Y -52.386,Z 160,A -25.8656,B 24.9659,C -1.3511,E1 25.1475,E2 472.5164} C_DIS
LIN {X 124.7799,Y -57.2799,Z 160,A -28.1704,B 24.9664,C -1.3397,E1 25.1449,E2 474.8354} C_DIS
LIN {X 123.2984,Y -60.4029,Z 160,A -29.6535,B 24.9667,C -1.3329,E1 25.1431,E2 476.3266} C_DIS
LIN {X 121.7956,Y -63.3793,Z 160,A -31.0717,B 24.967,C -1.3271,E1 25.1413,E2 477.7509} C_DIS
LIN {X 119.7009,Y -67.254,Z 160,A -32.8642,B 24.9672,C -1.3242,E1 25.1389,E2 479.5411} C_DIS
LIN {X 117.7354,Y -70.6396,Z 160,A -34.5284,B 24.9675,C -1.3175,E1 25.1365,E2 481.2123} C_DIS
LIN {X 115.4439,Y -74.3253,Z 160,A -36.436,B 24.968,C -1.3067,E1 25.1336,E2 483.1358} C_DIS
LIN {X 112.136,Y -79.2271,Z 160,A -38.7465,B 24.968,C -1.3086,E1 25.13,E2 485.4305} C_DIS
LIN {X 109.7283,Y -82.5298,Z 160,A -40.5044,B 24.9683,C -1.3008,E1 25.1271,E2 487.1983} C_DIS
LIN {X 107.0528,Y -85.972,Z 160,A -42.3191,B 24.9685,C -1.2961,E1 25.1239,E2 489.0157} C_DIS
LIN {X 104.2642,Y -89.3337,Z 160,A -44.1335,B 24.9688,C -1.2917,E1 25.1206,E2 490.8322} C_DIS
LIN {X 101.3023,Y -92.6788,Z 160,A -45.9855,B 24.969,C -1.2875,E1 25.1172,E2 492.6858} C_DIS
LIN {X 98.2127,Y -95.9466,Z 160,A -47.8563,B 24.9692,C -1.283,E1 25.1136,E2 494.5591} C_DIS
LIN {X 94.982,Y -99.1456,Z 160,A -49.7376,B 24.9694,C -1.2792,E1 25.1098,E2 496.4414} C_DIS
LIN {X 91.5692,Y -102.3058,Z 160,A -51.6297,B 24.9694,C -1.2773,E1 25.1059,E2 498.3305} C_DIS
LIN {X 88.1893,Y -105.2333,Z 160,A -53.4936,B 24.9696,C -1.2731,E1 25.1019,E2 500.197} C_DIS
LIN {X 84.6734,Y -108.0826,Z 160,A -55.3629,B 24.9698,C -1.2699,E1 25.0978,E2 502.0669} C_DIS
LIN {X 81.2536,Y -110.6764,Z 160,A -57.1743,B 24.97,C -1.2649,E1 25.0938,E2 503.8836} C_DIS
LIN {X 77.7195,Y -113.1861,Z 160,A -58.9552,B 24.9701,C -1.2626,E1 25.0897,E2 505.6637} C_DIS
LIN {X 73.9624,Y -115.6762,Z 160,A -60.6286,B 24.9698,C -1.2705,E1 25.0859,E2 507.3129} C_DIS
LIN {X 71.1719,Y -117.4138,Z 160,A -62.2158,B 24.9705,C -1.2558,E1 25.082,E2 508.93} C_DIS
LIN {X 67.2052,Y -119.7284,Z 160,A -64.0367,B 24.9704,C -1.2576,E1 25.0776,E2 510.7412} C_DIS
LIN {X 64.0588,Y -121.4388,Z 160,A -65.563,B 24.9706,C -1.2532,E1 25.0739,E2 512.2736} C_DIS
LIN {X 59.5738,Y -123.7013,Z 160,A -67.6356,B 24.9706,C -1.2509,E1 25.0687,E2 514.3458} C_DIS
LIN {X 56.3312,Y -125.2108,Z 160,A -69.1067,B 24.9707,C -1.2498,E1 25.0649,E2 515.816} C_DIS
LIN {X 51.8301,Y -127.1409,Z 160,A -71.0328,B 24.9706,C -1.2532,E1 25.06,E2 517.7294} C_DIS
LIN {X 45.7274,Y -129.4625,Z 160,A -73.8946,B 24.9711,C -1.2418,E1 25.0525,E2 520.6122} C_DIS
LIN {X 42.2271,Y -130.6445,Z 160,A -75.4341,B 24.9712,C -1.24,E1 25.0484,E2 522.153} C_DIS
LIN {X 38.5573,Y -131.7735,Z 160,A -76.9191,B 24.971,C -1.2446,E1 25.0445,E2 523.6245} C_DIS
LIN {X 34.0082,Y -133.0204,Z 160,A -78.9547,B 24.9713,C -1.2387,E1 25.0389,E2 525.6707} C_DIS
LIN {X 30.7822,Y -133.8037,Z 160,A -80.2776,B 24.9712,C -1.2408,E1 25.0354,E2 526.9869} C_DIS
LIN {X 27.8756,Y -134.4402,Z 160,A -81.6337,B 24.9715,C -1.2333,E1 25.0316,E2 528.3588} C_DIS
LIN {X 24.2098,Y -135.1475,Z 160,A -83.0926,B 24.9713,C -1.2375,E1 25.0276,E2 529.8062} C_DIS
LIN {X 20.2777,Y -135.7952,Z 160,A -85.556,B 24.9734,C -1.1926,E1 25.0206,E2 532.3735} C_DIS
LIN {X 14.5355,Y -136.5274,Z 160,A -87.2177,B 24.9716,C -1.2321,E1 25.0162,E2 533.9405} C_DIS
LIN {X 7.733,Y -137.0829,Z 160,A -90.1457,B 24.9718,C -1.2263,E1 25.008,E2 536.8808} C_DIS
LIN {X 4.2297,Y -137.2345,Z 160,A -91.6971,B 24.9721,C -1.2211,E1 25.0037,E2 538.4443} C_DIS
LIN {X 0.9739,Y -137.2937,Z 160,A -92.8756,B 24.9716,C -1.2305,E1 25.0004,E2 539.6002} C_DIS
Enddeposition()
LIN {X 0.9739,Y -137.2937,Z 160,A -92.8756,B 24.9716,C -1.2305,E1 25.0004,E2 539.6002} C_DIS
Startdeposition()
$VEL.CP = VEL_PRINT
LIN {X 1.7126,Y -136.3635,Z 160,A -91.0451,B 23.5685,C -1.0396,E1 23.5948,E2 538.0609} C_DIS
LIN {X 5.6231,Y -136.2575,Z 160,A -89.7141,B 23.5692,C -1.024,E1 23.5984,E2 536.7694} C_DIS
LIN {X 8.738,Y -136.0933,Z 160,A -87.9107,B 23.5681,C -1.0502,E1 23.6036,E2 534.9013} C_DIS
LIN {X 13.7493,Y -135.68,Z 160,A -86.4321,B 23.5694,C -1.0183,E1 23.6075,E2 533.5034} C_DIS
LIN {X 18.8392,Y -135.0662,Z 160,A -84.1905,B 23.5691,C -1.0242,E1 23.6138,E2 531.249} C_DIS
LIN {X 22.6417,Y -134.4803,Z 160,A -82.6091,B 23.5691,C -1.0235,E1 23.6181,E2 529.6708} C_DIS
LIN {X 26.7814,Y -133.7179,Z 160,A -80.8292,B 23.5691,C -1.0256,E1 23.623,E2 527.8879} C_DIS
LIN {X 30.1279,Y -133.0034,Z 160,A -79.4238,B 23.5691,C -1.0253,E1 23.6268,E2 526.4855} C_DIS
LIN {X 34.4236,Y -131.9587,Z 160,A -76.9488,B 23.5677,C -1.0596,E1 23.6337,E2 523.9286} C_DIS
LIN {X 39.332,Y -130.579,Z 160,A -75.3893,B 23.5689,C -1.0313,E1 23.6377,E2 522.4427} C_DIS
LIN {X 42.6807,Y -129.5224,Z 160,A -73.9388,B 23.5689,C -1.0318,E1 23.6416,E2 520.9939} C_DIS
LIN {X 49.0517,Y -127.2461,Z 160,A -71.1322,B 23.5688,C -1.0337,E1 23.6489,E2 518.1889} C_DIS
LIN {X 51.7499,Y -126.175,Z 160,A -69.6653,B 23.5681,C -1.0485,E1 23.6528,E2 516.6886} C_DIS
LIN {X 56.41,Y -124.1613,Z 160,A -67.6996,B 23.5684,C -1.0429,E1 23.6578,E2 514.7421} C_DIS
LIN {X 60.4519,Y -122.2418,Z 160,A -65.2412,B 23.5669,C -1.0769,E1 23.6641,E2 512.2059} C_DIS
LIN {X 65.3391,Y -119.703,Z 160,A -63.5169,B 23.5681,C -1.0493,E1 23.6682,E2 510.5556} C_DIS
LIN {X 69.3089,Y -117.4494,Z 160,A -61.8697,B 23.5686,C -1.0384,E1 23.6721,E2 508.9409} C_DIS
LIN {X 72.8047,Y -115.3147,Z 160,A -59.9307,B 23.5679,C -1.0533,E1 23.6768,E2 506.9713} C_DIS
LIN {X 76.6124,Y -112.821,Z 160,A -58.0144,B 23.5678,C -1.0573,E1 23.6812,E2 505.0518} C_DIS
LIN {X 80.3429,Y -110.196,Z 160,A -56.0614,B 23.5675,C -1.0633,E1 23.6857,E2 503.0913} C_DIS
LIN {X 83.8495,Y -107.5519,Z 160,A -54.2454,B 23.5675,C -1.0657,E1 23.6897,E2 501.2763} C_DIS
LIN {X 87.2846,Y -104.7834,Z 160,A -52.3934,B 23.5672,C -1.0698,E1 23.6937,E2 499.4217} C_DIS
LIN {X 90.4685,Y -102.0465,Z 160,A -50.6731,B 23.5672,C -1.0715,E1 23.6973,E2 497.7043} C_DIS
LIN {X 93.6943,Y -99.0929,Z 160,A -48.8494,B 23.567,C -1.0752,E1 23.701,E2 495.8795} C_DIS
LIN {X 96.9571,Y -95.9032,Z 160,A -46.921,B 23.5668,C -1.0805,E1 23.7049,E2 493.9465} C_DIS
LIN {X 100.0221,Y -92.7022,Z 160,A -45.0761,B 23.5666,C -1.0843,E1 23.7084,E2 492.1007} C_DIS
LIN {X 102.9428,Y -89.4475,Z 160,A -43.2449,B 23.5664,C -1.0888,E1 23.7118,E2 490.2672} C_DIS
LIN {X 105.7656,Y -86.0914,Z 160,A -41.4639,B 23.5664,C -1.0903,E1 23.7149,E2 488.4911} C_DIS
LIN {X 108.4259,Y -82.7155,Z 160,A -39.6274,B 23.5661,C -1.0969,E1 23.7181,E2 486.6474} C_DIS
LIN {X 111.136,Y -79.0374,Z 160,A -37.9325,B 23.5664,C -1.0901,E1 23.7208,E2 484.9783} C_DIS
LIN {X 114.3729,Y -74.2755,Z 160,A -35.5786,B 23.5662,C -1.0934,E1 23.7245,E2 482.6286} C_DIS
LIN {X 116.9722,Y -70.1115,Z 160,A -33.2221,B 23.5652,C -1.1153,E1 23.728,E2 480.2305} C_DIS
LIN {X 120.4174,Y -64.0125,Z 160,A -30.3666,B 23.5651,C -1.1192,E1 23.7319,E2 477.381} C_DIS
LIN {X 122.0525,Y -60.8356,Z 160,A -28.937,B 23.5651,C -1.1199,E1 23.7337,E2 475.9579} C_DIS
LIN {X 123.551,Y -57.7316,Z 160,A -27.6101,B 23.5651,C -1.1177,E1 23.7352,E2 474.6441} C_DIS
LIN {X 125.4566,Y -53.4661,Z 160,A -25.5561,B 23.5646,C -1.1287,E1 23.7376,E2 472.5747} C_DIS
LIN {X 128.1758,Y -46.568,Z 160,A -22.4334,B 23.5642,C -1.1388,E1 23.7407,E2 469.4454} C_DIS
LIN {X 129.2281,Y -43.5646,Z 160,A -20.7606,B 23.5631,C -1.1613,E1 23.7423,E2 467.7266} C_DIS
LIN {X 130.3383,Y -40.1186,Z 160,A -19.6208,B 23.5639,C -1.1454,E1 23.7432,E2 466.6334} C_DIS
LIN {X 131.3303,Y -36.7408,Z 160,A -18.1786,B 23.5638,C -1.1481,E1 23.7443,E2 465.1932} C_DIS
LIN {X 132.1813,Y -33.5505,Z 160,A -16.8368,B 23.5637,C -1.1501,E1 23.7452,E2 463.8547} C_DIS
LIN {X 132.89,Y -30.6245,Z 160,A -15.4517,B 23.5632,C -1.1607,E1 23.7461,E2 462.4517} C_DIS
LIN {X 133.6963,Y -26.8878,Z 160,A -13.8941,B 23.5631,C -1.1633,E1 23.747,E2 460.8974} C_DIS
LIN {X 134.4616,Y -22.7539,Z 160,A -12.1437,B 23.5628,C -1.1682,E1 23.7479,E2 459.1459} C_DIS
LIN {X 135.4739,Y -15.6417,Z 160,A -9.188,B 23.5625,C -1.1746,E1 23.749,E2 456.1928} C_DIS
LIN {X 135.8515,Y -11.9238,Z 160,A -7.5318,B 23.5621,C -1.1845,E1 23.7494,E2 454.5226} C_DIS
LIN {X 136.1312,Y -8.1226,Z 160,A -5.9916,B 23.562,C -1.1864,E1 23.7497,E2 452.9874} C_DIS
LIN {X 136.351,Y -2.4666,Z 160,A -3.2225,B 23.5606,C -1.2155,E1 23.7499,E2 450.1633} C_DIS
LIN {X 136.3642,Y 1.669,Z 160,A -1.8307,B 23.5612,C -1.2023,E1 23.7499,E2 448.8134} C_DIS
LIN {X 136.2689,Y 5.3292,Z 160,A 0.4287,B 23.559,C -1.2469,E1 23.7496,E2 446.4574} C_DIS
LIN {X 135.8846,Y 11.5318,Z 160,A 2.1877,B 23.5609,C -1.2086,E1 23.7493,E2 444.8046} C_DIS
LIN {X 135.4901,Y 15.5065,Z 160,A 3.9505,B 23.5604,C -1.2186,E1 23.7487,E2 443.0281} C_DIS
LIN {X 135.0106,Y 19.2281,Z 160,A 5.4045,B 23.5604,C -1.2171,E1 23.7482,E2 441.5872} C_DIS
LIN {X 134.4806,Y 22.6404,Z 160,A 6.8888,B 23.5602,C -1.2235,E1 23.7475,E2 440.0961} C_DIS
LIN {X 133.7278,Y 26.7328,Z 160,A 8.5747,B 23.5601,C -1.2257,E1 23.7466,E2 438.4154} C_DIS
LIN {X 133.0566,Y 29.8952,Z 160,A 9.9342,B 23.5599,C -1.23,E1 23.7458,E2 437.0534} C_DIS
LIN {X 132.2702,Y 33.2004,Z 160,A 11.3879,B 23.5596,C -1.2359,E1 23.7448,E2 435.5941} C_DIS
LIN {X 131.3531,Y 36.6591,Z 160,A 12.8972,B 23.5593,C -1.2409,E1 23.7437,E2 434.0815} C_DIS
LIN {X 128.1862,Y 46.5393,Z 160,A 17.2447,B 23.5587,C -1.2534,E1 23.74,E2 429.7292} C_DIS
LIN {X 126.2771,Y 51.4966,Z 160,A 19.5073,B 23.5583,C -1.2617,E1 23.7376,E2 427.4594} C_DIS
LIN {X 124.5685,Y 55.4997,Z 160,A 21.2155,B 23.5583,C -1.2606,E1 23.7357,E2 425.7641} C_DIS
LIN {X 123.1744,Y 58.5288,Z 160,A 22.6221,B 23.5581,C -1.2649,E1 23.7341,E2 424.3548} C_DIS
LIN {X 121.2357,Y 62.4483,Z 160,A 24.5322,B 23.5577,C -1.274,E1 23.7316,E2 422.4328} C_DIS
LIN {X 119.1613,Y 66.3225,Z 160,A 26.3745,B 23.5574,C -1.2789,E1 23.7292,E2 420.5886} C_DIS
LIN {X 116.9312,Y 70.1803,Z 160,A 28.1991,B 23.5573,C -1.2815,E1 23.7266,E2 418.7677} C_DIS
LIN {X 114.6367,Y 73.8688,Z 160,A 29.968,B 23.5572,C -1.2833,E1 23.724,E2 417.0038} C_DIS
LIN {X 109.249,Y 81.6254,Z 160,A 33.8419,B 23.5569,C -1.2883,E1 23.7178,E2 413.1376} C_DIS
LIN {X 106.7188,Y 84.9064,Z 160,A 35.7045,B 23.5564,C -1.2991,E1 23.7145,E2 411.2575} C_DIS
LIN {X 104.0709,Y 88.1324,Z 160,A 37.4779,B 23.5561,C -1.3044,E1 23.7113,E2 409.4798} C_DIS
LIN {X 100.2435,Y 92.4624,Z 160,A 39.8945,B 23.5558,C -1.3093,E1 23.7068,E2 407.0622} C_DIS
LIN {X 97.1015,Y 95.7572,Z 160,A 41.6854,B 23.5559,C -1.3071,E1 23.7034,E2 405.2851} C_DIS
LIN {X 93.4075,Y 99.3635,Z 160,A 43.862,B 23.5557,C -1.3121,E1 23.699,E2 403.1056} C_DIS
LIN {X 90.5694,Y 101.9573,Z 160,A 45.5544,B 23.5553,C -1.3195,E1 23.6954,E2 401.4021} C_DIS
LIN {X 82.901,Y 108.284,Z 160,A 49.6867,B 23.555,C -1.3251,E1 23.6865,E2 397.2726} C_DIS
LIN {X 79.1143,Y 111.081,Z 160,A 51.6237,B 23.555,C -1.3264,E1 23.6821,E2 395.3396} C_DIS
LIN {X 75.5523,Y 113.5337,Z 160,A 53.4757,B 23.5547,C -1.3313,E1 23.6778,E2 393.4821} C_DIS
LIN {X 71.1728,Y 116.3292,Z 160,A 55.6369,B 23.5545,C -1.3336,E1 23.6727,E2 391.3226} C_DIS
LIN {X 67.283,Y 118.6217,Z 160,A 57.5709,B 23.5543,C -1.3383,E1 23.668,E2 389.3829} C_DIS
LIN {X 63.6513,Y 120.607,Z 160,A 59.1644,B 23.5546,C -1.3332,E1 23.6641,E2 387.8071} C_DIS
LIN {X 60.6952,Y 122.1217,Z 160,A 60.5982,B 23.5544,C -1.337,E1 23.6606,E2 386.368} C_DIS
LIN {X 57.5374,Y 123.6407,Z 160,A 62.0527,B 23.5544,C -1.3379,E1 23.6569,E2 384.9153} C_DIS
LIN {X 54.4263,Y 125.0415,Z 160,A 63.5106,B 23.5542,C -1.3408,E1 23.6532,E2 383.4539} C_DIS
LIN {X 47.7595,Y 127.7362,Z 160,A 66.5093,B 23.5541,C -1.3427,E1 23.6454,E2 380.4575} C_DIS
LIN {X 43.1958,Y 129.3509,Z 160,A 68.5174,B 23.5541,C -1.3432,E1 23.6401,E2 378.4525} C_DIS
LIN {X 40.0751,Y 130.3516,Z 160,A 69.947,B 23.5538,C -1.347,E1 23.6363,E2 377.0162} C_DIS
LIN {X 36.6438,Y 131.3574,Z 160,A 71.3389,B 23.5541,C -1.3425,E1 23.6326,E2 375.6382} C_DIS
LIN {X 33.504,Y 132.1931,Z 160,A 72.7907,B 23.5538,C -1.3478,E1 23.6286,E2 374.1755} C_DIS
LIN {X 29.6976,Y 133.1017,Z 160,A 74.5192,B 23.5535,C -1.353,E1 23.6239,E2 372.4366} C_DIS
LIN {X 25.2541,Y 134.0146,Z 160,A 77.0608,B 23.5517,C -1.3864,E1 23.6167,E2 369.8146} C_DIS
LIN {X 19.6254,Y 134.9538,Z 160,A 78.75,B 23.5536,C -1.3509,E1 23.6123,E2 368.2158} C_DIS
LIN {X 15.8894,Y 135.4444,Z 160,A 80.3619,B 23.5536,C -1.3527,E1 23.6078,E2 366.6007} C_DIS
LIN {X 10.0797,Y 136.0001,Z 160,A 83.2668,B 23.5523,C -1.3759,E1 23.5996,E2 363.6395} C_DIS
LIN {X 5.574,Y 136.2594,Z 160,A 84.6464,B 23.5537,C -1.3497,E1 23.5959,E2 362.326} C_DIS
LIN {X 1.9981,Y 136.3588,Z 160,A 86.0417,B 23.554,C -1.3441,E1 23.592,E2 360.9448} C_DIS
LIN {X -3.0084,Y 136.3418,Z 160,A 88.6265,B 23.5527,C -1.3678,E1 23.5847,E2 358.3007} C_DIS
LIN {X -6.5971,Y 136.2136,Z 160,A 89.783,B 23.5537,C -1.3497,E1 23.5816,E2 357.1893} C_DIS
LIN {X -10.1465,Y 135.9952,Z 160,A 91.2861,B 23.5537,C -1.3495,E1 23.5774,E2 355.6861} C_DIS
LIN {X -14.3768,Y 135.6132,Z 160,A 93.0515,B 23.5537,C -1.3477,E1 23.5725,E2 353.9243} C_DIS
LIN {X -17.9267,Y 135.1897,Z 160,A 94.5704,B 23.5537,C -1.3477,E1 23.5683,E2 352.4042} C_DIS
LIN {X -21.9139,Y 134.6018,Z 160,A 96.2423,B 23.5539,C -1.3454,E1 23.5637,E2 350.7364} C_DIS
LIN {X -25.1885,Y 134.0271,Z 160,A 97.6295,B 23.5539,C -1.3438,E1 23.5598,E2 349.3515} C_DIS
LIN {X -28.6243,Y 133.335,Z 160,A 99.1485,B 23.5539,C -1.3449,E1 23.5557,E2 347.8279} C_DIS
LIN {X -32.587,Y 132.4237,Z 160,A 100.9178,B 23.5539,C -1.3463,E1 23.5509,E2 346.0526} C_DIS
LIN {X -36.1187,Y 131.5043,Z 160,A 103.108,B 23.5522,C -1.3773,E1 23.5448,E2 343.7811} C_DIS
LIN {X -41.4922,Y 129.9073,Z 160,A 105.1204,B 23.5533,C -1.3575,E1 23.5395,E2 341.8144} C_DIS
LIN {X -45.1748,Y 128.6741,Z 160,A 106.4905,B 23.5541,C -1.3426,E1 23.536,E2 340.4789} C_DIS
LIN {X -48.242,Y 127.5555,Z 160,A 108.1719,B 23.5533,C -1.356,E1 23.5315,E2 338.7601} C_DIS
LIN {X -52.0159,Y 126.0642,Z 160,A 109.5462,B 23.5543,C -1.3374,E1 23.5281,E2 337.4293} C_DIS
LIN {X -55.2904,Y 124.6621,Z 160,A 110.9851,B 23.5546,C -1.3324,E1 23.5244,E2 335.9993} C_DIS
LIN {X -58.5528,Y 123.1629,Z 160,A 112.279,B 23.5553,C -1.3196,E1 23.5212,E2 334.734} C_DIS
LIN {X -62.6811,Y 121.1165,Z 160,A 114.3917,B 23.555,C -1.325,E1 23.5159,E2 332.6018} C_DIS
LIN {X -67.889,Y 118.2761,Z 160,A 117.0145,B 23.555,C -1.3269,E1 23.5095,E2 329.966} C_DIS
LIN {X -72.0973,Y 115.7583,Z 160,A 119.5721,B 23.5538,C -1.3473,E1 23.5032,E2 327.3488} C_DIS
LIN {X -76.2039,Y 113.0976,Z 160,A 121.1934,B 23.5552,C -1.3221,E1 23.4996,E2 325.785} C_DIS
LIN {X -80.0745,Y 110.3906,Z 160,A 123.1158,B 23.5555,C -1.315,E1 23.4952,E2 323.8732} C_DIS
LIN {X -82.7911,Y 108.3681,Z 160,A 125.0089,B 23.5545,C -1.3347,E1 23.4909,E2 321.9232} C_DIS
LIN {X -86.4021,Y 105.5116,Z 160,A 126.5125,B 23.5558,C -1.3097,E1 23.4878,E2 320.4766} C_DIS
LIN {X -89.7083,Y 102.7153,Z 160,A 128.2786,B 23.5562,C -1.303,E1 23.4841,E2 318.72} C_DIS
LIN {X -92.8814,Y 99.8551,Z 160,A 130.1244,B 23.5562,C -1.3012,E1 23.4803,E2 316.8707} C_DIS
LIN {X -96.0607,Y 96.8006,Z 160,A 131.9782,B 23.5565,C -1.2968,E1 23.4766,E2 315.0196} C_DIS
LIN {X -98.9183,Y 93.8794,Z 160,A 133.7601,B 23.5565,C -1.2957,E1 23.4731,E2 313.2325} C_DIS
LIN {X -101.983,Y 90.5403,Z 160,A 135.6763,B 23.5568,C -1.2914,E1 23.4695,E2 311.3179} C_DIS
LIN {X -106.8027,Y 84.801,Z 160,A 138.5389,B 23.5579,C -1.2694,E1 23.4645,E2 308.4964} C_DIS
LIN {X -110.1892,Y 80.3523,Z 160,A 141.2107,B 23.5574,C -1.2783,E1 23.46,E2 305.7885} C_DIS
LIN {X -114.7489,Y 73.6935,Z 160,A 144.5976,B 23.5579,C -1.2686,E1 23.4547,E2 302.4081} C_DIS
LIN {X -117.1479,Y 69.8167,Z 160,A 146.4965,B 23.5583,C -1.2622,E1 23.4519,E2 300.5147} C_DIS
Enddeposition()
END
